    S364_M_FRT_PNL_제품감지_유 AT %MW2002.12 : BOOL;
    S364_M_FRT_PNL_제품감지_이상 AT %MW2014.3 : BOOL;
    S364_M_FRT_RACK_제품감지_무 AT %MW2002.7 : BOOL;
    S364_M_FRT_RACK_제품감지_유 AT %MW2002.6 : BOOL;
    S364_M_FRT_RACK_제품감지_이상 AT %MW2014.0 : BOOL;
    S364_M_LC_정상 AT %MW2007.5 : BOOL; (* S364_M_LC_정상 *)
    S364_M_LH_CB_OFF AT %MW2021.1 : BOOL; (* S364_M_LH_CB_OFF *)
    S364_M_LH_CP_OFF AT %MW2017.0 : BOOL; (* S364_M_LH_CP_OFF *)
    S364_M_LH_INV_이상 AT %MW2019.0 : BOOL; (* S364_M_LH_INV_이상 *)
    S364_M_LH_MC_이상 AT %MW2023.0 : BOOL; (* S364_M_LH_MC_이상 *)
    S364_M_LH_NFB_OFF AT %MW2021.0 : BOOL; (* S364_M_LH_NFB_OFF *)
    S364_M_LH_공기압_이상 AT %MW2013.0 : BOOL; (* S364_M_LH_공기압_이상 *)
    S364_M_MAT_정상 AT %MW2007.6 : BOOL; (* S364_M_MAT_정상 *)
    S364_M_OP_ESTOP_NORMAL AT %MW2007.1 : BOOL; (* S364_M_OP_ESTOP_NORMAL *)
    S364_M_OP_LC_이상 AT %MW2012.0 : BOOL; (* S364_M_OP_LC_이상 *)
    S364_M_OP_MAT_이상 AT %MW2012.1 : BOOL; (* S364_M_OP_MAT_이상 *)
    S364_M_R361_1_DATA_전송_MEMO AT %MW9012.8 : BOOL; (* S364 M R361 1 DATA 전송 MEMO *)
    S364_M_R361_1_DATA_전송_PLS AT %MW9012.9 : BOOL; (* S364 M R361 1 DATA 전송 PLS *)
    S364_M_R361_1_DATA_전송_SIGN AT %MW9012.10 : BOOL; (* S364 M R361 1 DATA 전송 SIGN *)
    S364_M_R361_1_DATA_전송_완료 AT %MW9012.11 : BOOL; (* S364 M R361 1 DATA 전송 완료 *)
    S364_M_R361_1_언로딩완료 AT %MW2001.4 : BOOL;
    S364_M_R361_2_로딩가능 AT %MW2004.9 : BOOL;
    S364_M_R361_2_로딩완료 AT %MW2001.2 : BOOL;
    S364_M_R364_1_용접가능 AT %MW2004.10 : BOOL;
    S364_M_R364_1_용접완료 AT %MW2001.3 : BOOL;
    S364_M_RH_CB_OFF AT %MW2021.4 : BOOL; (* S364_M_RH_CB_OFF *)
    S364_M_RH_CP_OFF AT %MW2017.1 : BOOL; (* S364_M_RH_CP_OFF *)
    S364_M_RH_INV_이상 AT %MW2019.1 : BOOL; (* S364_M_RH_INV_이상 *)
    S364_M_RH_MC_이상 AT %MW2023.1 : BOOL; (* S364_M_RH_MC_이상 *)
    S364_M_RH_NFB_OFF AT %MW2021.3 : BOOL; (* S364_M_RH_NFB_OFF *)
    S364_M_RH_공기압_이상 AT %MW2013.1 : BOOL; (* S364_M_RH_공기압_이상 *)
    S364_M_RR_PNL_제품감지_무 AT %MW2002.15 : BOOL;
    S364_M_RR_PNL_제품감지_유 AT %MW2002.14 : BOOL;
    S364_M_RR_PNL_제품감지_이상 AT %MW2014.4 : BOOL;
    S364_M_RR_RACK_제품감지_무 AT %MW2002.11 : BOOL;
    S364_M_RR_RACK_제품감지_유 AT %MW2002.10 : BOOL;
    S364_M_RR_RACK_제품감지_이상 AT %MW2014.2 : BOOL;
    S364_M_S102_간섭무 AT %MW2004.2 : BOOL; (* S364_M_S102_간섭무 *)
    S364_M_SAFETY_불간섭 AT %MW2004.4 : BOOL; (* S364_M_SAFETY_불간섭 *)
    S364_M_SEMI_자동모드 AT %MW2000.2 : BOOL; (* S364_M_SEMI_자동모드 *)
    S364_M_SEQ AT %MW10120 : WORD; (* S364 M SEQ *)
    S364_M_VIN_NO_1_2 AT %MW10131 : WORD; (* S364 M VIN NO 1 2 *)
    S364_M_VIN_NO_3_4 AT %MW10132 : WORD; (* S364 M VIN NO 3 4 *)
    S364_M_VIN_NO_5_6 AT %MW10133 : WORD; (* S364 M VIN NO 5 6 *)
    S364_M_VIN_NO_7_8 AT %MW10134 : WORD; (* S364 M VIN NO 7 8 *)
    S364_M_VIN_NO_9_10 AT %MW10135 : WORD; (* S364 M VIN NO 9 10 *)
    S364_M_공정_SAFETY_NORMAL AT %MW2007.7 : BOOL; (* S364_M_공정_SAFETY_NORMAL *)
    S364_M_공정_불간섭 AT %MW2004.1 : BOOL; (* S364_M_공정_불간섭 *)
    S364_M_공정_원위치 AT %MW2004.0 : BOOL; (* S364_M_공정_원위치 *)
    S364_M_공정_제품감지_무 AT %MW2002.5 : BOOL; (* S364_M_공정_제품감지_무 *)
    S364_M_공정_제품감지_유 AT %MW2002.4 : BOOL; (* S364_M_공정_제품감지_유 *)
    S364_M_공정_차종_AX AT %MW2002.3 : BOOL; (* S364_M_공정_차종_AX *)
    S364_M_공정_차종_무 AT %MW2002.1 : BOOL; (* S364_M_공정_차종_무 *)
    S364_M_공정_차종_보조 AT %MW2002.2 : BOOL; (* S364_M_공정_차종_보조 *)
    S364_M_공정_차종_유 AT %MW2002.0 : BOOL; (* S364_M_공정_차종_유 *)
    S364_M_동작_선택_1 AT %MW2040.0 : BOOL; (* S364_M_동작_선택_1 *)
    S364_M_동작_선택_10 AT %MW2040.9 : BOOL; (* S364_M_동작_선택_10 *)
    S364_M_동작_선택_11 AT %MW2040.10 : BOOL; (* S364_M_동작_선택_11 *)
    S364_M_동작_선택_12 AT %MW2040.11 : BOOL; (* S364_M_동작_선택_12 *)
    S364_M_동작_선택_13 AT %MW2040.12 : BOOL; (* S364_M_동작_선택_13 *)
    S364_M_동작_선택_14 AT %MW2040.13 : BOOL; (* S364_M_동작_선택_14 *)
    S364_M_동작_선택_15 AT %MW2040.14 : BOOL; (* S364_M_동작_선택_15 *)
    S364_M_동작_선택_16 AT %MW2040.15 : BOOL; (* S364_M_동작_선택_16 *)
    S364_M_동작_선택_17 AT %MW2041.0 : BOOL; (* S364_M_동작_선택_17 *)
    S364_M_동작_선택_18 AT %MW2041.1 : BOOL; (* S364_M_동작_선택_18 *)
    S364_M_동작_선택_19 AT %MW2041.2 : BOOL; (* S364_M_동작_선택_19 *)
    S364_M_동작_선택_2 AT %MW2040.1 : BOOL; (* S364_M_동작_선택_2 *)
    S364_M_동작_선택_20 AT %MW2041.3 : BOOL; (* S364_M_동작_선택_20 *)
    S364_M_동작_선택_21 AT %MW2041.4 : BOOL; (* S364_M_동작_선택_21 *)
    S364_M_동작_선택_22 AT %MW2041.5 : BOOL; (* S364_M_동작_선택_22 *)
    S364_M_동작_선택_23 AT %MW2041.6 : BOOL; (* S364_M_동작_선택_23 *)
    S364_M_동작_선택_24 AT %MW2041.7 : BOOL; (* S364_M_동작_선택_24 *)
    S364_M_동작_선택_25 AT %MW2041.8 : BOOL; (* S364_M_동작_선택_25 *)
    S364_M_동작_선택_26 AT %MW2041.9 : BOOL; (* S364_M_동작_선택_26 *)
    S364_M_동작_선택_27 AT %MW2041.10 : BOOL; (* S364_M_동작_선택_27 *)
    S364_M_동작_선택_28 AT %MW2041.11 : BOOL; (* S364_M_동작_선택_28 *)
    S364_M_동작_선택_29 AT %MW2041.12 : BOOL; (* S364_M_동작_선택_29 *)
    S364_M_동작_선택_3 AT %MW2040.2 : BOOL; (* S364_M_동작_선택_3 *)
    S364_M_동작_선택_30 AT %MW2041.13 : BOOL; (* S364_M_동작_선택_30 *)
    S364_M_동작_선택_31 AT %MW2041.14 : BOOL; (* S364_M_동작_선택_31 *)
    S364_M_동작_선택_32 AT %MW2041.15 : BOOL; (* S364_M_동작_선택_32 *)
    S364_M_동작_선택_4 AT %MW2040.3 : BOOL; (* S364_M_동작_선택_4 *)
    S364_M_동작_선택_5 AT %MW2040.4 : BOOL; (* S364_M_동작_선택_5 *)
    S364_M_동작_선택_6 AT %MW2040.5 : BOOL; (* S364_M_동작_선택_6 *)
    S364_M_동작_선택_7 AT %MW2040.6 : BOOL; (* S364_M_동작_선택_7 *)
    S364_M_동작_선택_8 AT %MW2040.7 : BOOL; (* S364_M_동작_선택_8 *)
    S364_M_동작_선택_9 AT %MW2040.8 : BOOL; (* S364_M_동작_선택_9 *)
    S364_M_부저_정지_보조 AT %MW2000.11 : BOOL; (* S364_M_부저_정지_보조 *)
    S364_M_수동모드 AT %MW2000.3 : BOOL; (* S364 선택 수동모드 *)
    S364_M_운전준비_ON AT %MW2000.0 : BOOL; (* S364 운전준비 ON *)
    S364_M_이상_리셋_보조 AT %MW2000.10 : BOOL; (* S364_M_이상_리셋_보조 *)
    S364_M_자동_START AT %MW2000.5 : BOOL; (* S364 자동운전중 *)
    S364_M_자동_운전중 AT %MW2000.4 : BOOL; (* S364 자동운전중 *)
    S364_M_자동모드 AT %MW2000.1 : BOOL; (* S364 선택 자동모드 *)
    S364_M_작업_완료 AT %MW2001.0 : BOOL; (* S364_M_작업_완료 *)
    S364_M_작업완료_SET_PLS AT %MW2000.8 : BOOL; (* S364 M 작업완료 SET PLS *)
    S364_M_작업완료_리셋_PLS AT %MW2000.9 : BOOL; (* S364 M 작업완료 리셋 PLS *)
    S364_M_작업자_작업가능 AT %MW2004.8 : BOOL;
    S364_M_작업자_작업완료 AT %MW2001.1 : BOOL;
    S364_M_전체_용접완료 AT %MW2006.0 : BOOL;
    S364_M_차종1_AX AT %MW10121.0 : BOOL; (* S364 M 차종1 AX *)
    S364_M_차종1_B AT %MW10121.1 : BOOL; (* S364 M 차종1 B *)
    S364_M_차종1_C AT %MW10121.2 : BOOL; (* S364 M 차종1 C *)
    S364_M_차종1_D AT %MW10121.3 : BOOL; (* S364 M 차종1 D *)
    S364_M_차종1_E AT %MW10121.4 : BOOL; (* S364 M 차종1 E *)
    S364_M_차종1_F AT %MW10121.5 : BOOL; (* S364 M 차종1 F *)
    S364_M_차종1_G AT %MW10121.6 : BOOL; (* S364 M 차종1 G *)
    S364_M_차종1_H AT %MW10121.7 : BOOL; (* S364 M 차종1 H *)
    S364_M_차종2_3DR AT %MW10121.8 : BOOL; (* S364 M 차종2 3DR *)
    S364_M_차종2_4DR AT %MW10121.9 : BOOL; (* S364 M 차종2 4DR *)
    S364_M_차종2_5DR AT %MW10121.10 : BOOL; (* S364 M 차종2 5DR *)
    S364_M_차종2_SP1 AT %MW10121.12 : BOOL; (* S364 M 차종2 SP1 *)
    S364_M_차종2_SP2 AT %MW10121.13 : BOOL; (* S364 M 차종2 SP2 *)
    S364_M_차종2_WGN AT %MW10121.11 : BOOL; (* S364 M 차종2 WGN *)
    S364_M_차종3_LHD AT %MW10121.14 : BOOL; (* S364 M 차종3 LHD *)
    S364_M_차종3_RHD AT %MW10121.15 : BOOL; (* S364 M 차종3 RHD *)
    S364_M_차종4_EEC AT %MW10122.3 : BOOL; (* S364 M 차종4 EEC *)
    S364_M_차종4_SP1 AT %MW10122.8 : BOOL; (* S364 M 차종4 SP1 *)
    S364_M_차종4_SP2 AT %MW10122.9 : BOOL; (* S364 M 차종4 SP2 *)
    S364_M_차종4_SP3 AT %MW10122.11 : BOOL; (* S364 M 차종4 SP3 *)
    S364_M_차종4_SP4 AT %MW10122.12 : BOOL; (* S364 M 차종4 SP4 *)
    S364_M_차종4_SP5 AT %MW10122.13 : BOOL; (* S364 M 차종4 SP5 *)
    S364_M_차종4_SP6 AT %MW10122.14 : BOOL; (* S364 M 차종4 SP6 *)
    S364_M_차종4_SP7 AT %MW10122.15 : BOOL; (* S364 M 차종4 SP7 *)
    S364_M_차종4_내수 AT %MW10122.0 : BOOL; (* S364 M 차종4 내수 *)
    S364_M_차종4_러시아 AT %MW10122.10 : BOOL; (* S364 M 차종4 러시아 *)
    S364_M_차종4_북미 AT %MW10122.2 : BOOL; (* S364 M 차종4 북미 *)
    S364_M_차종4_브라질 AT %MW10122.7 : BOOL; (* S364 M 차종4 브라질 *)
    S364_M_차종4_수출 AT %MW10122.1 : BOOL; (* S364 M 차종4 수출 *)
    S364_M_차종4_중국 AT %MW10122.6 : BOOL; (* S364 M 차종4 중국 *)
    S364_M_차종4_중동 AT %MW10122.5 : BOOL; (* S364 M 차종4 중동 *)
    S364_M_차종4_호주 AT %MW10122.4 : BOOL; (* S364 M 차종4 호주 *)
    S364_M_차종5_AT AT %MW10123.1 : BOOL; (* S364 M 차종5 AT *)
    S364_M_차종5_MT AT %MW10123.0 : BOOL; (* S364 M 차종5 MT *)
    S364_M_차종5_SP1 AT %MW10123.2 : BOOL; (* S364 M 차종5 SP1 *)
    S364_M_차종6_DSROOF AT %MW10123.6 : BOOL; (* S364 M 차종6 DSROOF *)
    S364_M_차종6_SP1 AT %MW10123.7 : BOOL; (* S364 M 차종6 SP1 *)
    S364_M_차종6_썬루프 AT %MW10123.4 : BOOL; (* S364 M 차종6 썬루프 *)
    S364_M_차종6_일반루프 AT %MW10123.3 : BOOL; (* S364 M 차종6 일반루프 *)
    S364_M_차종6_파노라마루프 AT %MW10123.5 : BOOL; (* S364 M 차종6 파노라마루프 *)
    S364_M_차종7_DSL AT %MW10123.9 : BOOL; (* S364 M 차종7 DSL *)
    S364_M_차종7_GSL AT %MW10123.8 : BOOL; (* S364 M 차종7 GSL *)
    S364_M_차종7_SP1 AT %MW10123.10 : BOOL; (* S364 M 차종7 SP1 *)
    S364_M_차종7_SP2 AT %MW10123.11 : BOOL; (* S364 M 차종7 SP2 *)
    S364_M_차종7_SP3 AT %MW10123.12 : BOOL; (* S364 M 차종7 SP3 *)
    S364_M_차종7_SP4 AT %MW10123.13 : BOOL; (* S364 M 차종7 SP4 *)
    S364_M_차종7_SP5 AT %MW10123.14 : BOOL; (* S364 M 차종7 SP5 *)
    S364_M_차종7_SP6 AT %MW10123.15 : BOOL; (* S364 M 차종7 SP6 *)
    S364_M_차종8_2WD AT %MW10124.0 : BOOL; (* S364 M 차종8 2WD *)
    S364_M_차종8_4WD AT %MW10124.1 : BOOL; (* S364 M 차종8 4WD *)
    S364_M_차종8_SP1 AT %MW10124.2 : BOOL; (* S364 M 차종8 SP1 *)
    S364_M_차종9_MPI AT %MW10124.3 : BOOL; (* S364 M 차종9 MPI *)
    S364_M_차종9_SP1 AT %MW10124.5 : BOOL; (* S364 M 차종9 SP1 *)
    S364_M_차종9_SP10 AT %MW10124.14 : BOOL; (* S364 M 차종9 SP10 *)
    S364_M_차종9_SP11 AT %MW10124.15 : BOOL; (* S364 M 차종9 SP11 *)
    S364_M_차종9_SP2 AT %MW10124.6 : BOOL; (* S364 M 차종9 SP2 *)
    S364_M_차종9_SP3 AT %MW10124.7 : BOOL; (* S364 M 차종9 SP3 *)
    S364_M_차종9_SP4 AT %MW10124.8 : BOOL; (* S364 M 차종9 SP4 *)
    S364_M_차종9_SP5 AT %MW10124.9 : BOOL; (* S364 M 차종9 SP5 *)
    S364_M_차종9_SP6 AT %MW10124.10 : BOOL; (* S364 M 차종9 SP6 *)
    S364_M_차종9_SP7 AT %MW10124.11 : BOOL; (* S364 M 차종9 SP7 *)
    S364_M_차종9_SP8 AT %MW10124.12 : BOOL; (* S364 M 차종9 SP8 *)
    S364_M_차종9_SP9 AT %MW10124.13 : BOOL; (* S364 M 차종9 SP9 *)
    S364_M_차종9_T_GDI AT %MW10124.4 : BOOL; (* S364 M 차종9 T GDI *)
    S364_M_차종_AS AT %MW10130.9 : BOOL; (* S364 M 차종 AS *)
    S364_M_차종_OPT1_R_RACK_무 AT %MW10125.3 : BOOL; (* S364 M 차종 OPT1 R RACK 무 *)
    S364_M_차종_OPT1_R_RACK_유 AT %MW10125.2 : BOOL; (* S364 M 차종 OPT1 R RACK 유 *)
    S364_M_차종_OPT1_SP1 AT %MW10125.10 : BOOL; (* S364 M 차종 OPT1 SP1 *)
    S364_M_차종_OPT1_SP2 AT %MW10125.11 : BOOL; (* S364 M 차종 OPT1 SP2 *)
    S364_M_차종_OPT1_SP3 AT %MW10125.12 : BOOL; (* S364 M 차종 OPT1 SP3 *)
    S364_M_차종_OPT1_SP4 AT %MW10125.13 : BOOL; (* S364 M 차종 OPT1 SP4 *)
    S364_M_차종_OPT1_SP5 AT %MW10125.14 : BOOL; (* S364 M 차종 OPT1 SP5 *)
    S364_M_차종_OPT1_SP6 AT %MW10125.15 : BOOL; (* S364 M 차종 OPT1 SP6 *)
    S364_M_차종_OPT1_S_REP_EATER_무 AT %MW10125.7 : BOOL; (* S364 M 차종 OPT1 S REP EATER 무 *)
    S364_M_차종_OPT1_S_REP_EATER_유 AT %MW10125.6 : BOOL; (* S364 M 차종 OPT1 S REP EATER 유 *)
    S364_M_차종_OPT1_VAN_무 AT %MW10125.9 : BOOL; (* S364 M 차종 OPT1 VAN 무 *)
    S364_M_차종_OPT1_VAN_유 AT %MW10125.8 : BOOL; (* S364 M 차종 OPT1 VAN 유 *)
    S364_M_차종_OPT1_슬라이딩_무 AT %MW10125.1 : BOOL; (* S364 M 차종 OPT1 슬라이딩 무 *)
    S364_M_차종_OPT1_슬라이딩_유 AT %MW10125.0 : BOOL; (* S364 M 차종 OPT1 슬라이딩 유 *)
    S364_M_차종_OPT1_폴딩_무 AT %MW10125.5 : BOOL; (* S364 M 차종 OPT1 폴딩 무 *)
    S364_M_차종_OPT1_폴딩_유 AT %MW10125.4 : BOOL; (* S364 M 차종 OPT1 폴딩 유 *)
    S364_M_차종_OPT2_SP_WORD1 AT %MW10126 : WORD; (* S364 M 차종 OPT2 SP WORD1 *)
    S364_M_차종_OPT3_SP_WORD2 AT %MW10127 : WORD; (* S364 M 차종 OPT3 SP WORD2 *)
    S364_M_차종_OPT4_SP_WORD3 AT %MW10128 : WORD; (* S364 M 차종 OPT4 SP WORD3 *)
    S364_M_차종_OPT5_SP_WORD4 AT %MW10129 : WORD; (* S364 M 차종 OPT5 SP WORD4 *)
    S364_M_차종_SP1 AT %MW10130.0 : BOOL; (* S364 M 차종 SP1 *)
    S364_M_차종_SP2 AT %MW10130.1 : BOOL; (* S364 M 차종 SP2 *)
    S364_M_차종_SP3 AT %MW10130.2 : BOOL; (* S364 M 차종 SP3 *)
    S364_M_차종_SP4 AT %MW10130.3 : BOOL; (* S364 M 차종 SP4 *)
    S364_M_차종_SP5 AT %MW10130.4 : BOOL; (* S364 M 차종 SP5 *)
    S364_M_차종_SP6 AT %MW10130.5 : BOOL; (* S364 M 차종 SP6 *)
    S364_M_차종_SP7 AT %MW10130.6 : BOOL; (* S364 M 차종 SP7 *)
    S364_M_차종_SP8 AT %MW10130.7 : BOOL; (* S364 M 차종 SP8 *)
    S364_M_차종_SP9 AT %MW10130.15 : BOOL; (* S364 M 차종 SP9 *)
    S364_M_차종_공대차 AT %MW10130.12 : BOOL; (* S364 M 차종 공대차 *)
    S364_M_차종_공차 AT %MW10130.10 : BOOL; (* S364 M 차종 공차 *)
    S364_M_차종_불량대차 AT %MW10130.13 : BOOL; (* S364 M 차종 불량대차 *)
    S364_M_차종_불량차 AT %MW10130.11 : BOOL; (* S364 M 차종 불량차 *)
    S364_M_차종_비축 AT %MW10130.8 : BOOL; (* S364 M 차종 비축 *)
    S364_M_차종_취출대차 AT %MW10130.14 : BOOL; (* S364 M 차종 취출대차 *)
    S364_M_총괄_CP_이상 AT %MW2009.7 : BOOL; (* S364 CP OFF 이상 *)
    S364_M_총괄_CT_이상 AT %MW2010.4 : BOOL; (* S364   TACK TIME 이상 *)
    S364_M_총괄_EOCR_이상 AT %MW2009.8 : BOOL; (* S364_M_총괄_EOCR_이상 *)
    S364_M_총괄_INV_이상 AT %MW2009.9 : BOOL; (* S364_M_총괄_INV_이상 *)
    S364_M_총괄_LS_이상 AT %MW2009.15 : BOOL; (* S364 LS 이상 *)
    S364_M_총괄_MATCH_이상 AT %MW2010.0 : BOOL; (* S364 매트SW 이상 *)
    S364_M_총괄_MC_이상 AT %MW2009.13 : BOOL; (* S364_M_총괄_MC_이상 *)
    S364_M_총괄_MOTOR_이상 AT %MW2010.3 : BOOL; (* S364_M_총괄_MOTOR_이상 *)
    S364_M_총괄_NFB_이상 AT %MW2009.11 : BOOL; (* S364_M_총괄_NFB_이상 *)
    S364_M_총괄_ROBOT_이상 AT %MW2010.1 : BOOL; (* S364 ROBOT 이상 *)
    S364_M_총괄_SAFETY_이상 AT %MW2009.2 : BOOL; (* S364 SAFETY 이상 *)
    S364_M_총괄_SRV_이상 AT %MW2009.10 : BOOL; (* S364_M_총괄_SRV_이상 *)
    S364_M_총괄_공기압_이상 AT %MW2009.3 : BOOL; (* S364 공기압 이상 *)
    S364_M_총괄_비상정지_이상 AT %MW2009.1 : BOOL; (* S364_M_총괄_비상정지_이상 *)
    S364_M_총괄_사양_이상 AT %MW2009.6 : BOOL; (* S364 사양 이상 *)
    S364_M_총괄_오버런_이상 AT %MW2009.12 : BOOL; (* S364_M_총괄_오버런_이상 *)
    S364_M_총괄_용접타점수_이상 AT %MW2010.2 : BOOL; (* S364 용접타점수 이상 *)
    S364_M_총괄_이상 AT %MW2009.0 : BOOL; (* S364_M_총괄_이상 *)
    S364_M_총괄_제품감지_이상 AT %MW2009.4 : BOOL; (* S364 제품감지 이상 *)
    S364_M_총괄_차종_이상 AT %MW2009.5 : BOOL; (* S364 차종 이상 *)
    S364_M_총괄_통신_이상 AT %MW2009.14 : BOOL; (* S364 통신이상 *)
    S364_RH_M_NODE_7_15_통신_이상 AT %MW2024.1 : BOOL;
    S364_전진_ON AT %MW2048.1 : BOOL; (* S364_전진_ON *)
    S364_후진_ON AT %MW2048.2 : BOOL; (* S364_후진_ON *)
    S365_HOME AT %MW2548.0 : BOOL; (* S365_HOME *)
    S365_M_BYPASS_보조 AT %MW2503.15 : BOOL; (* S365 M BYPASS 보조 *)
    S365_M_CTIME_OVER_ALRAM AT %MW2507.14 : BOOL; (* S365_M_CTIME_OVER_ALRAM *)
    S365_M_CTIME_OVER_MUTE AT %MW2507.13 : BOOL; (* S365_M_CTIME_OVER_MUTE *)
    S365_M_DATA_삭제_PLS AT %MW9013.0 : BOOL; (* S365 M DATA 삭제 PLS *)
    S365_M_DATA_삭제_SIGN AT %MW9013.1 : BOOL; (* S365 M DATA 삭제 SIGN *)
    S365_M_DATA_삭제_완료 AT %MW9013.2 : BOOL; (* S365 M DATA 삭제 완료 *)
    S365_M_LC_정상 AT %MW2507.5 : BOOL; (* S365_M_LC_정상 *)
    S365_M_MAT_정상 AT %MW2507.6 : BOOL; (* S365_M_MAT_정상 *)
    S365_M_NODE_6_01_통신_이상 AT %MW2524.0 : BOOL;
    S365_M_OP_ESTOP_NORMAL AT %MW2507.1 : BOOL; (* S365_M_OP_ESTOP_NORMAL *)
    S365_M_R361_1_안착완료 AT %MW2501.1 : BOOL;
    S365_M_R361_1_언로딩완료 AT %MW2501.2 : BOOL;
    S365_M_S102_간섭무 AT %MW2504.2 : BOOL; (* S365_M_S102_간섭무 *)
    S365_M_S361_1_DATA_전송_MEMO AT %MW9013.8 : BOOL; (* S365 M S361 1 DATA 전송 MEMO *)
    S365_M_S361_1_DATA_전송_PLS AT %MW9013.9 : BOOL; (* S365 M S361 1 DATA 전송 PLS *)
    S365_M_S361_1_DATA_전송_SIGN AT %MW9013.10 : BOOL; (* S365 M S361 1 DATA 전송 SIGN *)
    S365_M_S361_1_DATA_전송_완료 AT %MW9013.11 : BOOL; (* S365 M S361 1 DATA 전송 완료 *)
    S365_M_SAFETY_불간섭 AT %MW2504.4 : BOOL; (* S365_M_SAFETY_불간섭 *)
    S365_M_SEMI_자동모드 AT %MW2500.2 : BOOL; (* S365_M_SEMI_자동모드 *)
    S365_M_SEQ AT %MW10140 : WORD; (* S365 M SEQ *)
    S365_M_VIN_NO_1_2 AT %MW10151 : WORD; (* S365 M VIN NO 1 2 *)
    S365_M_VIN_NO_3_4 AT %MW10152 : WORD; (* S365 M VIN NO 3 4 *)
    S365_M_VIN_NO_5_6 AT %MW10153 : WORD; (* S365 M VIN NO 5 6 *)
    S365_M_VIN_NO_7_8 AT %MW10154 : WORD; (* S365 M VIN NO 7 8 *)
    S365_M_VIN_NO_9_10 AT %MW10155 : WORD; (* S365 M VIN NO 9 10 *)
    S365_M_공정_SAFETY_NORMAL AT %MW2507.7 : BOOL; (* S365_M_공정_SAFETY_NORMAL *)
    S365_M_공정_불간섭 AT %MW2504.1 : BOOL; (* S365_M_공정_불간섭 *)
    S365_M_공정_원위치 AT %MW2504.0 : BOOL; (* S365_M_공정_원위치 *)
    S365_M_공정_제품감지_무 AT %MW2501.4 : BOOL; (* S365_M_공정_제품감지_무 *)
    S365_M_공정_제품감지_유 AT %MW2501.3 : BOOL; (* S365_M_공정_제품감지_유 *)
    S365_M_공정_차종_무 AT %MW2502.1 : BOOL; (* S365_M_공정_차종_무 *)
    S365_M_공정_차종_보조 AT %MW2502.2 : BOOL; (* S365_M_공정_차종_보조 *)
    S365_M_공정_차종_유 AT %MW2502.0 : BOOL; (* S365_M_공정_차종_유 *)
    S365_M_동작_선택_1 AT %MW2540.0 : BOOL; (* S365_M_동작_선택_1 *)
    S365_M_동작_선택_10 AT %MW2540.9 : BOOL; (* S365_M_동작_선택_10 *)
    S365_M_동작_선택_11 AT %MW2540.10 : BOOL; (* S365_M_동작_선택_11 *)
    S365_M_동작_선택_12 AT %MW2540.11 : BOOL; (* S365_M_동작_선택_12 *)
    S365_M_동작_선택_13 AT %MW2540.12 : BOOL; (* S365_M_동작_선택_13 *)
    S365_M_동작_선택_14 AT %MW2540.13 : BOOL; (* S365_M_동작_선택_14 *)
    S365_M_동작_선택_15 AT %MW2540.14 : BOOL; (* S365_M_동작_선택_15 *)
    S365_M_동작_선택_16 AT %MW2540.15 : BOOL; (* S365_M_동작_선택_16 *)
    S365_M_동작_선택_17 AT %MW2541.0 : BOOL; (* S365_M_동작_선택_17 *)
    S365_M_동작_선택_18 AT %MW2541.1 : BOOL; (* S365_M_동작_선택_18 *)
    S365_M_동작_선택_19 AT %MW2541.2 : BOOL; (* S365_M_동작_선택_19 *)
    S365_M_동작_선택_2 AT %MW2540.1 : BOOL; (* S365_M_동작_선택_2 *)
    S365_M_동작_선택_20 AT %MW2541.3 : BOOL; (* S365_M_동작_선택_20 *)
    S365_M_동작_선택_21 AT %MW2541.4 : BOOL; (* S365_M_동작_선택_21 *)
    S365_M_동작_선택_22 AT %MW2541.5 : BOOL; (* S365_M_동작_선택_22 *)
    S365_M_동작_선택_23 AT %MW2541.6 : BOOL; (* S365_M_동작_선택_23 *)
    S365_M_동작_선택_24 AT %MW2541.7 : BOOL; (* S365_M_동작_선택_24 *)
    S365_M_동작_선택_25 AT %MW2541.8 : BOOL; (* S365_M_동작_선택_25 *)
    S365_M_동작_선택_26 AT %MW2541.9 : BOOL; (* S365_M_동작_선택_26 *)
    S365_M_동작_선택_27 AT %MW2541.10 : BOOL; (* S365_M_동작_선택_27 *)
    S365_M_동작_선택_28 AT %MW2541.11 : BOOL; (* S365_M_동작_선택_28 *)
    S365_M_동작_선택_29 AT %MW2541.12 : BOOL; (* S365_M_동작_선택_29 *)
    S365_M_동작_선택_3 AT %MW2540.2 : BOOL; (* S365_M_동작_선택_3 *)
    S365_M_동작_선택_30 AT %MW2541.13 : BOOL; (* S365_M_동작_선택_30 *)
    S365_M_동작_선택_31 AT %MW2541.14 : BOOL; (* S365_M_동작_선택_31 *)
    S365_M_동작_선택_32 AT %MW2541.15 : BOOL; (* S365_M_동작_선택_32 *)
    S365_M_동작_선택_4 AT %MW2540.3 : BOOL; (* S365_M_동작_선택_4 *)
    S365_M_동작_선택_5 AT %MW2540.4 : BOOL; (* S365_M_동작_선택_5 *)
    S365_M_동작_선택_6 AT %MW2540.5 : BOOL; (* S365_M_동작_선택_6 *)
    S365_M_동작_선택_7 AT %MW2540.6 : BOOL; (* S365_M_동작_선택_7 *)
    S365_M_동작_선택_8 AT %MW2540.7 : BOOL; (* S365_M_동작_선택_8 *)
    S365_M_동작_선택_9 AT %MW2540.8 : BOOL; (* S365_M_동작_선택_9 *)
    S365_M_부저_정지_보조 AT %MW2500.11 : BOOL; (* S365_M_부저_정지_보조 *)
    S365_M_수동모드 AT %MW2500.3 : BOOL; (* S365 선택 수동모드 *)
    S365_M_운전준비_ON AT %MW2500.0 : BOOL; (* S365 운전준비 ON *)
    S365_M_이상_리셋_보조 AT %MW2500.10 : BOOL; (* S365_M_이상_리셋_보조 *)
    S365_M_자동_START AT %MW2500.5 : BOOL; (* S365 자동운전중 *)
    S365_M_자동_운전중 AT %MW2500.4 : BOOL; (* S365 자동운전중 *)
    S365_M_자동모드 AT %MW2500.1 : BOOL; (* S365 선택 자동모드 *)
    S365_M_작업_완료 AT %MW2501.0 : BOOL; (* S365_M_작업_완료 *)
    S365_M_작업완료_SET_PLS AT %MW2500.8 : BOOL; (* S365 M 작업완료 SET PLS *)
    S365_M_작업완료_리셋_PLS AT %MW2500.9 : BOOL; (* S365 M 작업완료 리셋 PLS *)
    S365_M_차종1_AX AT %MW10141.0 : BOOL; (* S365 M 차종1 AX *)
    S365_M_차종1_B AT %MW10141.1 : BOOL; (* S365 M 차종1 B *)
    S365_M_차종1_C AT %MW10141.2 : BOOL; (* S365 M 차종1 C *)
    S365_M_차종1_D AT %MW10141.3 : BOOL; (* S365 M 차종1 D *)
    S365_M_차종1_E AT %MW10141.4 : BOOL; (* S365 M 차종1 E *)
    S365_M_차종1_F AT %MW10141.5 : BOOL; (* S365 M 차종1 F *)
    S365_M_차종1_G AT %MW10141.6 : BOOL; (* S365 M 차종1 G *)
    S365_M_차종1_H AT %MW10141.7 : BOOL; (* S365 M 차종1 H *)
    S365_M_차종2_3DR AT %MW10141.8 : BOOL; (* S365 M 차종2 3DR *)
    S365_M_차종2_4DR AT %MW10141.9 : BOOL; (* S365 M 차종2 4DR *)
    S365_M_차종2_5DR AT %MW10141.10 : BOOL; (* S365 M 차종2 5DR *)
    S365_M_차종2_SP1 AT %MW10141.12 : BOOL; (* S365 M 차종2 SP1 *)
    S365_M_차종2_SP2 AT %MW10141.13 : BOOL; (* S365 M 차종2 SP2 *)
    S365_M_차종2_WGN AT %MW10141.11 : BOOL; (* S365 M 차종2 WGN *)
    S365_M_차종3_LHD AT %MW10141.14 : BOOL; (* S365 M 차종3 LHD *)
    S365_M_차종3_RHD AT %MW10141.15 : BOOL; (* S365 M 차종3 RHD *)
    S365_M_차종4_EEC AT %MW10142.3 : BOOL; (* S365 M 차종4 EEC *)
    S365_M_차종4_SP1 AT %MW10142.8 : BOOL; (* S365 M 차종4 SP1 *)
    S365_M_차종4_SP2 AT %MW10142.9 : BOOL; (* S365 M 차종4 SP2 *)
    S365_M_차종4_SP3 AT %MW10142.11 : BOOL; (* S365 M 차종4 SP3 *)
    S365_M_차종4_SP4 AT %MW10142.12 : BOOL; (* S365 M 차종4 SP4 *)
    S365_M_차종4_SP5 AT %MW10142.13 : BOOL; (* S365 M 차종4 SP5 *)
    S365_M_차종4_SP6 AT %MW10142.14 : BOOL; (* S365 M 차종4 SP6 *)
    S365_M_차종4_SP7 AT %MW10142.15 : BOOL; (* S365 M 차종4 SP7 *)
    S365_M_차종4_내수 AT %MW10142.0 : BOOL; (* S365 M 차종4 내수 *)
    S365_M_차종4_러시아 AT %MW10142.10 : BOOL; (* S365 M 차종4 러시아 *)
    S365_M_차종4_북미 AT %MW10142.2 : BOOL; (* S365 M 차종4 북미 *)
    S365_M_차종4_브라질 AT %MW10142.7 : BOOL; (* S365 M 차종4 브라질 *)
    S365_M_차종4_수출 AT %MW10142.1 : BOOL; (* S365 M 차종4 수출 *)
    S365_M_차종4_중국 AT %MW10142.6 : BOOL; (* S365 M 차종4 중국 *)
    S365_M_차종4_중동 AT %MW10142.5 : BOOL; (* S365 M 차종4 중동 *)
    S365_M_차종4_호주 AT %MW10142.4 : BOOL; (* S365 M 차종4 호주 *)
    S365_M_차종5_AT AT %MW10143.1 : BOOL; (* S365 M 차종5 AT *)
    S365_M_차종5_MT AT %MW10143.0 : BOOL; (* S365 M 차종5 MT *)
    S365_M_차종5_SP1 AT %MW10143.2 : BOOL; (* S365 M 차종5 SP1 *)
    S365_M_차종6_DSROOF AT %MW10143.6 : BOOL; (* S365 M 차종6 DSROOF *)
    S365_M_차종6_SP1 AT %MW10143.7 : BOOL; (* S365 M 차종6 SP1 *)
    S365_M_차종6_썬루프 AT %MW10143.4 : BOOL; (* S365 M 차종6 썬루프 *)
    S365_M_차종6_일반루프 AT %MW10143.3 : BOOL; (* S365 M 차종6 일반루프 *)
    S365_M_차종6_파노라마루프 AT %MW10143.5 : BOOL; (* S365 M 차종6 파노라마루프 *)
    S365_M_차종7_DSL AT %MW10143.9 : BOOL; (* S365 M 차종7 DSL *)
    S365_M_차종7_GSL AT %MW10143.8 : BOOL; (* S365 M 차종7 GSL *)
    S365_M_차종7_SP1 AT %MW10143.10 : BOOL; (* S365 M 차종7 SP1 *)
    S365_M_차종7_SP2 AT %MW10143.11 : BOOL; (* S365 M 차종7 SP2 *)
    S365_M_차종7_SP3 AT %MW10143.12 : BOOL; (* S365 M 차종7 SP3 *)
    S365_M_차종7_SP4 AT %MW10143.13 : BOOL; (* S365 M 차종7 SP4 *)
    S365_M_차종7_SP5 AT %MW10143.14 : BOOL; (* S365 M 차종7 SP5 *)
    S365_M_차종7_SP6 AT %MW10143.15 : BOOL; (* S365 M 차종7 SP6 *)
    S365_M_차종8_2WD AT %MW10144.0 : BOOL; (* S365 M 차종8 2WD *)
    S365_M_차종8_4WD AT %MW10144.1 : BOOL; (* S365 M 차종8 4WD *)
    S365_M_차종8_SP1 AT %MW10144.2 : BOOL; (* S365 M 차종8 SP1 *)
    S365_M_차종9_MPI AT %MW10144.3 : BOOL; (* S365 M 차종9 MPI *)
    S365_M_차종9_SP1 AT %MW10144.5 : BOOL; (* S365 M 차종9 SP1 *)
    S365_M_차종9_SP10 AT %MW10144.14 : BOOL; (* S365 M 차종9 SP10 *)
    S365_M_차종9_SP11 AT %MW10144.15 : BOOL; (* S365 M 차종9 SP11 *)
    S365_M_차종9_SP2 AT %MW10144.6 : BOOL; (* S365 M 차종9 SP2 *)
    S365_M_차종9_SP3 AT %MW10144.7 : BOOL; (* S365 M 차종9 SP3 *)
    S365_M_차종9_SP4 AT %MW10144.8 : BOOL; (* S365 M 차종9 SP4 *)
    S365_M_차종9_SP5 AT %MW10144.9 : BOOL; (* S365 M 차종9 SP5 *)
    S365_M_차종9_SP6 AT %MW10144.10 : BOOL; (* S365 M 차종9 SP6 *)
    S365_M_차종9_SP7 AT %MW10144.11 : BOOL; (* S365 M 차종9 SP7 *)
    S365_M_차종9_SP8 AT %MW10144.12 : BOOL; (* S365 M 차종9 SP8 *)
    S365_M_차종9_SP9 AT %MW10144.13 : BOOL; (* S365 M 차종9 SP9 *)
    S365_M_차종9_T_GDI AT %MW10144.4 : BOOL; (* S365 M 차종9 T GDI *)
    S365_M_차종_AS AT %MW10150.9 : BOOL; (* S365 M 차종 AS *)
    S365_M_차종_OPT1_R_RACK_무 AT %MW10145.3 : BOOL; (* S365 M 차종 OPT1 R RACK 무 *)
    S365_M_차종_OPT1_R_RACK_유 AT %MW10145.2 : BOOL; (* S365 M 차종 OPT1 R RACK 유 *)
    S365_M_차종_OPT1_SP1 AT %MW10145.10 : BOOL; (* S365 M 차종 OPT1 SP1 *)
    S365_M_차종_OPT1_SP2 AT %MW10145.11 : BOOL; (* S365 M 차종 OPT1 SP2 *)
    S365_M_차종_OPT1_SP3 AT %MW10145.12 : BOOL; (* S365 M 차종 OPT1 SP3 *)
    S365_M_차종_OPT1_SP4 AT %MW10145.13 : BOOL; (* S365 M 차종 OPT1 SP4 *)
    S365_M_차종_OPT1_SP5 AT %MW10145.14 : BOOL; (* S365 M 차종 OPT1 SP5 *)
    S365_M_차종_OPT1_SP6 AT %MW10145.15 : BOOL; (* S365 M 차종 OPT1 SP6 *)
    S365_M_차종_OPT1_S_REP_EATER_무 AT %MW10145.7 : BOOL; (* S365 M 차종 OPT1 S REP EATER 무 *)
    S365_M_차종_OPT1_S_REP_EATER_유 AT %MW10145.6 : BOOL; (* S365 M 차종 OPT1 S REP EATER 유 *)
    S365_M_차종_OPT1_VAN_무 AT %MW10145.9 : BOOL; (* S365 M 차종 OPT1 VAN 무 *)
    S365_M_차종_OPT1_VAN_유 AT %MW10145.8 : BOOL; (* S365 M 차종 OPT1 VAN 유 *)
    S365_M_차종_OPT1_슬라이딩_무 AT %MW10145.1 : BOOL; (* S365 M 차종 OPT1 슬라이딩 무 *)
    S365_M_차종_OPT1_슬라이딩_유 AT %MW10145.0 : BOOL; (* S365 M 차종 OPT1 슬라이딩 유 *)
    S365_M_차종_OPT1_폴딩_무 AT %MW10145.5 : BOOL; (* S365 M 차종 OPT1 폴딩 무 *)
    S365_M_차종_OPT1_폴딩_유 AT %MW10145.4 : BOOL; (* S365 M 차종 OPT1 폴딩 유 *)
    S365_M_차종_OPT2_SP_WORD1 AT %MW10146 : WORD; (* S365 M 차종 OPT2 SP WORD1 *)
    S365_M_차종_OPT3_SP_WORD2 AT %MW10147 : WORD; (* S365 M 차종 OPT3 SP WORD2 *)
    S365_M_차종_OPT4_SP_WORD3 AT %MW10148 : WORD; (* S365 M 차종 OPT4 SP WORD3 *)
    S365_M_차종_OPT5_SP_WORD4 AT %MW10149 : WORD; (* S365 M 차종 OPT5 SP WORD4 *)
    S365_M_차종_SP1 AT %MW10150.0 : BOOL; (* S365 M 차종 SP1 *)
    S365_M_차종_SP2 AT %MW10150.1 : BOOL; (* S365 M 차종 SP2 *)
    S365_M_차종_SP3 AT %MW10150.2 : BOOL; (* S365 M 차종 SP3 *)
    S365_M_차종_SP4 AT %MW10150.3 : BOOL; (* S365 M 차종 SP4 *)
    S365_M_차종_SP5 AT %MW10150.4 : BOOL; (* S365 M 차종 SP5 *)
    S365_M_차종_SP6 AT %MW10150.5 : BOOL; (* S365 M 차종 SP6 *)
    S365_M_차종_SP7 AT %MW10150.6 : BOOL; (* S365 M 차종 SP7 *)
    S365_M_차종_SP8 AT %MW10150.7 : BOOL; (* S365 M 차종 SP8 *)
    S365_M_차종_SP9 AT %MW10150.15 : BOOL; (* S365 M 차종 SP9 *)
    S365_M_차종_공대차 AT %MW10150.12 : BOOL; (* S365 M 차종 공대차 *)
    S365_M_차종_공차 AT %MW10150.10 : BOOL; (* S365 M 차종 공차 *)
    S365_M_차종_불량대차 AT %MW10150.13 : BOOL; (* S365 M 차종 불량대차 *)
    S365_M_차종_불량차 AT %MW10150.11 : BOOL; (* S365 M 차종 불량차 *)
    S365_M_차종_비축 AT %MW10150.8 : BOOL; (* S365 M 차종 비축 *)
    S365_M_차종_취출대차 AT %MW10150.14 : BOOL; (* S365 M 차종 취출대차 *)
    S365_M_총괄_CP_이상 AT %MW2509.7 : BOOL; (* S365 CP OFF 이상 *)
    S365_M_총괄_CT_이상 AT %MW2510.4 : BOOL; (* S365   TACK TIME 이상 *)
    S365_M_총괄_EOCR_이상 AT %MW2509.8 : BOOL; (* S365_M_총괄_EOCR_이상 *)
    S365_M_총괄_INV_이상 AT %MW2509.9 : BOOL; (* S365_M_총괄_INV_이상 *)
    S365_M_총괄_LS_이상 AT %MW2509.15 : BOOL; (* S365 LS 이상 *)
    S365_M_총괄_MATCH_이상 AT %MW2510.0 : BOOL; (* S365 매트SW 이상 *)
    S365_M_총괄_MC_이상 AT %MW2509.13 : BOOL; (* S365_M_총괄_MC_이상 *)
    S365_M_총괄_MOTOR_이상 AT %MW2510.3 : BOOL; (* S365_M_총괄_MOTOR_이상 *)
    S365_M_총괄_NFB_이상 AT %MW2509.11 : BOOL; (* S365_M_총괄_NFB_이상 *)
    S365_M_총괄_ROBOT_이상 AT %MW2510.1 : BOOL; (* S365 ROBOT 이상 *)
    S365_M_총괄_SAFETY_이상 AT %MW2509.2 : BOOL; (* S365 SAFETY 이상 *)
    S365_M_총괄_SRV_이상 AT %MW2509.10 : BOOL; (* S365_M_총괄_SRV_이상 *)
    S365_M_총괄_공기압_이상 AT %MW2509.3 : BOOL; (* S365 공기압 이상 *)
    S365_M_총괄_비상정지_이상 AT %MW2509.1 : BOOL; (* S365_M_총괄_비상정지_이상 *)
    S365_M_총괄_사양_이상 AT %MW2509.6 : BOOL; (* S365 사양 이상 *)
    S365_M_총괄_오버런_이상 AT %MW2509.12 : BOOL; (* S365_M_총괄_오버런_이상 *)
    S365_M_총괄_용접타점수_이상 AT %MW2510.2 : BOOL; (* S365 용접타점수 이상 *)
    S365_M_총괄_이상 AT %MW2509.0 : BOOL; (* S365_M_총괄_이상 *)
    S365_M_총괄_제품감지_이상 AT %MW2509.4 : BOOL; (* S365 제품감지 이상 *)
    S365_M_총괄_차종_이상 AT %MW2509.5 : BOOL; (* S365 차종 이상 *)
    S365_M_총괄_통신_이상 AT %MW2509.14 : BOOL; (* S365 통신이상 *)
    S365_전진_ON AT %MW2548.1 : BOOL; (* S365_전진_ON *)
    S365_후진_ON AT %MW2548.2 : BOOL; (* S365_후진_ON *)
    S366_HOME AT %MW3048.0 : BOOL; (* S366_HOME *)
    S366_LH_M_NODE_8_10_통신_이상 AT %MW3024.1 : BOOL;
    S366_M_AX_LH_CLP_전진_LS_이상 AT %MW3104.5 : BOOL; (* S366_M_AX_LH_CLP_전진_LS_이상 *)
    S366_M_AX_LH_CLP_전진_보조 AT %MW3104.1 : BOOL; (* S366_M_AX_LH_CLP_전진_보조 *)
    S366_M_AX_LH_CLP_전진단 AT %MW3104.3 : BOOL; (* S366_M_AX_LH_CLP_전진단 *)
    S366_M_AX_LH_CLP_조건 AT %MW3104.0 : BOOL; (* S366_M_AX_LH_CLP_조건 *)
    S366_M_AX_LH_CLP_후진_LS_이상 AT %MW3104.6 : BOOL; (* S366_M_AX_LH_CLP_후진_LS_이상 *)
    S366_M_AX_LH_CLP_후진_보조 AT %MW3104.2 : BOOL; (* S366_M_AX_LH_CLP_후진_보조 *)
    S366_M_AX_LH_CLP_후진단 AT %MW3104.4 : BOOL; (* S366_M_AX_LH_CLP_후진단 *)
    S366_M_AX_RH_CLP_전진_LS_이상 AT %MW3112.5 : BOOL; (* S366_M_AX_RH_CLP_전진_LS_이상 *)
    S366_M_AX_RH_CLP_전진_보조 AT %MW3112.1 : BOOL; (* S366_M_AX_RH_CLP_전진_보조 *)
    S366_M_AX_RH_CLP_전진단 AT %MW3112.3 : BOOL; (* S366_M_AX_RH_CLP_전진단 *)
    S366_M_AX_RH_CLP_조건 AT %MW3112.0 : BOOL; (* S366_M_AX_RH_CLP_조건 *)
    S366_M_AX_RH_CLP_후진_LS_이상 AT %MW3112.6 : BOOL; (* S366_M_AX_RH_CLP_후진_LS_이상 *)
    S366_M_AX_RH_CLP_후진_보조 AT %MW3112.2 : BOOL; (* S366_M_AX_RH_CLP_후진_보조 *)
    S366_M_AX_RH_CLP_후진단 AT %MW3112.4 : BOOL; (* S366_M_AX_RH_CLP_후진단 *)
    S366_M_BYPASS_보조 AT %MW3003.15 : BOOL; (* S366 M BYPASS 보조 *)
    S366_M_CP_OFF AT %MW3017.0 : BOOL;
    S366_M_CTIME_OVER_ALRAM AT %MW3007.14 : BOOL; (* S366_M_CTIME_OVER_ALRAM *)
    S366_M_CTIME_OVER_MUTE AT %MW3007.13 : BOOL; (* S366_M_CTIME_OVER_MUTE *)
    S366_M_DATA_삭제_PLS AT %MW9014.0 : BOOL; (* S366 M DATA 삭제 PLS *)
    S366_M_DATA_삭제_SIGN AT %MW9014.1 : BOOL; (* S366 M DATA 삭제 SIGN *)
    S366_M_DATA_삭제_완료 AT %MW9014.2 : BOOL; (* S366 M DATA 삭제 완료 *)
    S366_M_LC_정상 AT %MW3007.5 : BOOL; (* S366_M_LC_정상 *)
    S366_M_LH_CB_OFF AT %MW3021.2 : BOOL;
    S366_M_LH_CP_OFF AT %MW3017.2 : BOOL; (* S366_M_LH_CP_OFF *)
    S366_M_LH_INV_이상 AT %MW3019.0 : BOOL; (* S366_M_LH_INV_이상 *)
    S366_M_LH_MAIN_BAR_이상 AT %MW3012.0 : BOOL; (* S366_M_LH_MAIN_BAR_이상 *)
    S366_M_LH_MC_이상 AT %MW3023.0 : BOOL; (* S366_M_LH_MC_이상 *)
    S366_M_LH_NFB_OFF AT %MW3021.0 : BOOL; (* S366_M_LH_NFB_OFF *)
    S366_M_LH_STEP_MOVE_리셋_PLS AT %MW3101.14 : BOOL; (* S366_M_LH_STEP_MOVE_리셋_PLS *)
    S366_M_LH_TURN_1_포지션단 AT %MW3101.3 : BOOL; (* S366_M_LH_TURN_1_포지션단 *)
    S366_M_LH_TURN_2_포지션단 AT %MW3101.4 : BOOL; (* S366_M_LH_TURN_2_포지션단 *)
    S366_M_LH_TURN_3_포지션단 AT %MW3101.5 : BOOL; (* S366_M_LH_TURN_3_포지션단 *)
    S366_M_LH_TURN_4_포지션단 AT %MW3101.6 : BOOL; (* S366_M_LH_TURN_4_포지션단 *)
    S366_M_LH_TURN_LS_이상 AT %MW3101.7 : BOOL; (* S366_M_LH_TURN_LS_이상 *)
    S366_M_LH_TURN_MOVE_완료 AT %MW3101.8 : BOOL; (* S366_M_LH_TURN_MOVE_완료 *)
    S366_M_LH_TURN_수동_STEP_전진_보조 AT %MW3101.11 : BOOL; (* S366_M_LH_TURN_수동_STEP_전진_보조 *)
    S366_M_LH_TURN_수동_STEP_후진_보조 AT %MW3101.12 : BOOL; (* S366_M_LH_TURN_수동_STEP_후진_보조 *)
    S366_M_LH_TURN_수동_전진_보조 AT %MW3101.9 : BOOL; (* S366_M_LH_TURN_수동_전진_보조 *)
    S366_M_LH_TURN_수동_후진_보조 AT %MW3101.10 : BOOL; (* S366_M_LH_TURN_수동_후진_보조 *)
    S366_M_LH_TURN_전진_보조 AT %MW3101.1 : BOOL; (* S366_M_LH_TURN_전진_보조 *)
    S366_M_LH_TURN_조건 AT %MW3101.0 : BOOL; (* S366_M_LH_TURN_조건 *)
    S366_M_LH_TURN_후진_보조 AT %MW3101.2 : BOOL; (* S366_M_LH_TURN_후진_보조 *)
    S366_M_LH_공기압_이상 AT %MW3013.0 : BOOL; (* S366_M_LH_공기압_이상 *)
    S366_M_LH_자동_MOVE_리셋_PLS AT %MW3101.13 : BOOL; (* S366_M_LH_자동_MOVE_리셋_PLS *)
    S366_M_MAT_정상 AT %MW3007.6 : BOOL; (* S366_M_MAT_정상 *)
    S366_M_NODE_6_10_통신_이상 AT %MW3024.0 : BOOL;
    S366_M_OP_ESTOP_NORMAL AT %MW3007.1 : BOOL; (* S366_M_OP_ESTOP_NORMAL *)
    S366_M_R361_1_DATA_전송_MEMO AT %MW9014.8 : BOOL; (* S366 M R361 1 DATA 전송 MEMO *)
    S366_M_R361_1_DATA_전송_PLS AT %MW9014.9 : BOOL; (* S366 M R361 1 DATA 전송 PLS *)
    S366_M_R361_1_DATA_전송_SIGN AT %MW9014.10 : BOOL; (* S366 M R361 1 DATA 전송 SIGN *)
    S366_M_R361_1_DATA_전송_완료 AT %MW9014.11 : BOOL; (* S366 M R361 1 DATA 전송 완료 *)
    S366_M_R361_1_ROOF_로딩완료 AT %MW3001.2 : BOOL;
    S366_M_R361_1_동일차종_OK AT %MW3005.8 : BOOL;
    S366_M_R361_1_언로딩완료 AT %MW3001.4 : BOOL;
    S366_M_R361_1_차종매칭_조건 AT %MW3005.0 : BOOL;
    S366_M_R363_2_RAIL_로딩완료 AT %MW3001.1 : BOOL;
    S366_M_R366_1_용접가능 AT %MW3004.10 : BOOL;
    S366_M_R366_1_용접완료 AT %MW3001.3 : BOOL;
    S366_M_RAIL_로딩가능 AT %MW3004.8 : BOOL;
    S366_M_RH_CB_OFF AT %MW3021.3 : BOOL;
    S366_M_RH_CP_OFF AT %MW3017.3 : BOOL; (* S366_M_RH_CP_OFF *)
    S366_M_RH_INV_이상 AT %MW3019.1 : BOOL; (* S366_M_RH_INV_이상 *)
    S366_M_RH_MAIN_BAR_이상 AT %MW3012.1 : BOOL; (* S366_M_RH_MAIN_BAR_이상 *)
    S366_M_RH_MC_이상 AT %MW3023.1 : BOOL; (* S366_M_RH_MC_이상 *)
    S366_M_RH_NFB_OFF AT %MW3021.1 : BOOL; (* S366_M_RH_NFB_OFF *)
    S366_M_RH_STEP_MOVE_리셋_PLS AT %MW3109.14 : BOOL; (* S366_M_RH_STEP_MOVE_리셋_PLS *)
    S366_M_RH_TURN_1_포지션단 AT %MW3109.3 : BOOL; (* S366_M_RH_TURN_1_포지션단 *)
    S366_M_RH_TURN_2_포지션단 AT %MW3109.4 : BOOL; (* S366_M_RH_TURN_2_포지션단 *)
    S366_M_RH_TURN_3_포지션단 AT %MW3109.5 : BOOL; (* S366_M_RH_TURN_3_포지션단 *)
    S366_M_RH_TURN_4_포지션단 AT %MW3109.6 : BOOL; (* S366_M_RH_TURN_4_포지션단 *)
    S366_M_RH_TURN_LS_이상 AT %MW3109.7 : BOOL; (* S366_M_RH_TURN_LS_이상 *)
    S366_M_RH_TURN_MOVE_완료 AT %MW3109.8 : BOOL; (* S366_M_RH_TURN_MOVE_완료 *)
    S366_M_RH_TURN_수동_STEP_전진_보조 AT %MW3109.11 : BOOL; (* S366_M_RH_TURN_수동_STEP_전진_보조 *)
    S366_M_RH_TURN_수동_STEP_후진_보조 AT %MW3109.12 : BOOL; (* S366_M_RH_TURN_수동_STEP_후진_보조 *)
    S366_M_RH_TURN_수동_전진_보조 AT %MW3109.9 : BOOL; (* S366_M_RH_TURN_수동_전진_보조 *)
    S366_M_RH_TURN_수동_후진_보조 AT %MW3109.10 : BOOL; (* S366_M_RH_TURN_수동_후진_보조 *)
    S366_M_RH_TURN_전진_보조 AT %MW3109.1 : BOOL; (* S366_M_RH_TURN_전진_보조 *)
    S366_M_RH_TURN_조건 AT %MW3109.0 : BOOL; (* S366_M_RH_TURN_조건 *)
    S366_M_RH_TURN_후진_보조 AT %MW3109.2 : BOOL; (* S366_M_RH_TURN_후진_보조 *)
    S366_M_RH_공기압_이상 AT %MW3013.1 : BOOL; (* S366_M_RH_공기압_이상 *)
    S366_M_RH_자동_MOVE_리셋_PLS AT %MW3109.13 : BOOL; (* S366_M_RH_자동_MOVE_리셋_PLS *)
    S366_M_ROOF_로딩가능 AT %MW3004.9 : BOOL;
    S366_M_SAFETY_불간섭 AT %MW3004.4 : BOOL; (* S366_M_SAFETY_불간섭 *)
    S366_M_SEMI_자동모드 AT %MW3000.2 : BOOL; (* S366_M_SEMI_자동모드 *)
    S366_M_SEQ AT %MW10160 : WORD; (* S366 M SEQ *)
    S366_M_TURN_LOCK_전진_LS_이상 AT %MW3100.5 : BOOL; (* S366_M_TURN_LOCK_전진_LS_이상 *)
    S366_M_TURN_LOCK_전진_보조 AT %MW3100.1 : BOOL; (* S366_M_TURN_LOCK_전진_보조 *)
    S366_M_TURN_LOCK_전진단 AT %MW3100.3 : BOOL; (* S366_M_TURN_LOCK_전진단 *)
    S366_M_TURN_LOCK_조건 AT %MW3100.0 : BOOL; (* S366_M_TURN_LOCK_조건 *)
    S366_M_TURN_LOCK_후진_LS_이상 AT %MW3100.6 : BOOL; (* S366_M_TURN_LOCK_후진_LS_이상 *)
    S366_M_TURN_LOCK_후진_보조 AT %MW3100.2 : BOOL; (* S366_M_TURN_LOCK_후진_보조 *)
    S366_M_TURN_LOCK_후진단 AT %MW3100.4 : BOOL; (* S366_M_TURN_LOCK_후진단 *)
    S366_M_VIN_NO_1_2 AT %MW10171 : WORD; (* S366 M VIN NO 1 2 *)
    S366_M_VIN_NO_3_4 AT %MW10172 : WORD; (* S366 M VIN NO 3 4 *)
    S366_M_VIN_NO_5_6 AT %MW10173 : WORD; (* S366 M VIN NO 5 6 *)
    S366_M_VIN_NO_7_8 AT %MW10174 : WORD; (* S366 M VIN NO 7 8 *)
    S366_M_VIN_NO_9_10 AT %MW10175 : WORD; (* S366 M VIN NO 9 10 *)
    S366_M_공정_AX_FRT_PNL_제품감지_이상 AT %MW3014.4 : BOOL;
    S366_M_공정_AX_RAIL_제품감지_이상 AT %MW3014.3 : BOOL;
    S366_M_공정_AX_RR_PNL_제품감지_이상 AT %MW3014.5 : BOOL;
    S366_M_공정_AX_공용_제품감지_이상 AT %MW3014.0 : BOOL;
    S366_M_공정_AX_썬루프_제품감지_이상 AT %MW3014.2 : BOOL;
    S366_M_공정_AX_일반루프_제품감지_이상 AT %MW3014.1 : BOOL;
    S366_M_공정_FRT_PNL_제품감지_무 AT %MW3002.13 : BOOL;
    S366_M_공정_FRT_PNL_제품감지_유 AT %MW3002.12 : BOOL;
    S366_M_공정_RAIL_제품감지_무 AT %MW3001.15 : BOOL;
    S366_M_공정_RAIL_제품감지_유 AT %MW3001.14 : BOOL;
    S366_M_공정_RR_PNL_제품감지_무 AT %MW3002.15 : BOOL;
    S366_M_공정_RR_PNL_제품감지_유 AT %MW3002.14 : BOOL;
    S366_M_공정_SAFETY_NORMAL AT %MW3007.7 : BOOL; (* S366_M_공정_SAFETY_NORMAL *)
    S366_M_공정_공용_제품감지_무 AT %MW3001.9 : BOOL;
    S366_M_공정_공용_제품감지_유 AT %MW3001.8 : BOOL;
    S366_M_공정_불간섭 AT %MW3004.1 : BOOL; (* S366_M_공정_불간섭 *)
    S366_M_공정_썬루프_제품감지_무 AT %MW3001.13 : BOOL;
    S366_M_공정_썬루프_제품감지_유 AT %MW3001.12 : BOOL;
    S366_M_공정_원위치 AT %MW3004.0 : BOOL; (* S366_M_공정_원위치 *)
    S366_M_공정_일반루프_제품감지_무 AT %MW3001.11 : BOOL;
    S366_M_공정_일반루프_제품감지_유 AT %MW3001.10 : BOOL;
    S366_M_공정_제품감지_무 AT %MW3001.7 : BOOL; (* S366_M_공정_제품감지_무 *)
    S366_M_공정_제품감지_유 AT %MW3001.6 : BOOL; (* S366_M_공정_제품감지_유 *)
    S366_M_공정_차종_AX AT %MW3002.3 : BOOL; (* S366_M_공정_차종_AX *)
    S366_M_공정_차종_무 AT %MW3002.1 : BOOL; (* S366_M_공정_차종_무 *)
    S366_M_공정_차종_유 AT %MW3002.0 : BOOL; (* S366_M_공정_차종_유 *)
    S366_M_동작_선택_1 AT %MW3040.0 : BOOL; (* S366_M_동작_선택_1 *)
    S366_M_동작_선택_10 AT %MW3040.9 : BOOL; (* S366_M_동작_선택_10 *)
    S366_M_동작_선택_11 AT %MW3040.10 : BOOL; (* S366_M_동작_선택_11 *)
    S366_M_동작_선택_12 AT %MW3040.11 : BOOL; (* S366_M_동작_선택_12 *)
    S366_M_동작_선택_13 AT %MW3040.12 : BOOL; (* S366_M_동작_선택_13 *)
    S366_M_동작_선택_14 AT %MW3040.13 : BOOL; (* S366_M_동작_선택_14 *)
    S366_M_동작_선택_15 AT %MW3040.14 : BOOL; (* S366_M_동작_선택_15 *)
    S366_M_동작_선택_16 AT %MW3040.15 : BOOL; (* S366_M_동작_선택_16 *)
    S366_M_동작_선택_17 AT %MW3041.0 : BOOL; (* S366_M_동작_선택_17 *)
    S366_M_동작_선택_18 AT %MW3041.1 : BOOL; (* S366_M_동작_선택_18 *)
    S366_M_동작_선택_19 AT %MW3041.2 : BOOL; (* S366_M_동작_선택_19 *)
    S366_M_동작_선택_2 AT %MW3040.1 : BOOL; (* S366_M_동작_선택_2 *)
    S366_M_동작_선택_20 AT %MW3041.3 : BOOL; (* S366_M_동작_선택_20 *)
    S366_M_동작_선택_21 AT %MW3041.4 : BOOL; (* S366_M_동작_선택_21 *)
    S366_M_동작_선택_22 AT %MW3041.5 : BOOL; (* S366_M_동작_선택_22 *)
    S366_M_동작_선택_23 AT %MW3041.6 : BOOL; (* S366_M_동작_선택_23 *)
    S366_M_동작_선택_24 AT %MW3041.7 : BOOL; (* S366_M_동작_선택_24 *)
    S366_M_동작_선택_25 AT %MW3041.8 : BOOL; (* S366_M_동작_선택_25 *)
    S366_M_동작_선택_26 AT %MW3041.9 : BOOL; (* S366_M_동작_선택_26 *)
    S366_M_동작_선택_27 AT %MW3041.10 : BOOL; (* S366_M_동작_선택_27 *)
    S366_M_동작_선택_28 AT %MW3041.11 : BOOL; (* S366_M_동작_선택_28 *)
    S366_M_동작_선택_29 AT %MW3041.12 : BOOL; (* S366_M_동작_선택_29 *)
    S366_M_동작_선택_3 AT %MW3040.2 : BOOL; (* S366_M_동작_선택_3 *)
    S366_M_동작_선택_30 AT %MW3041.13 : BOOL; (* S366_M_동작_선택_30 *)
    S366_M_동작_선택_31 AT %MW3041.14 : BOOL; (* S366_M_동작_선택_31 *)
    S366_M_동작_선택_32 AT %MW3041.15 : BOOL; (* S366_M_동작_선택_32 *)
    S366_M_동작_선택_4 AT %MW3040.3 : BOOL; (* S366_M_동작_선택_4 *)
    S366_M_동작_선택_5 AT %MW3040.4 : BOOL; (* S366_M_동작_선택_5 *)
    S366_M_동작_선택_6 AT %MW3040.5 : BOOL; (* S366_M_동작_선택_6 *)
    S366_M_동작_선택_7 AT %MW3040.6 : BOOL; (* S366_M_동작_선택_7 *)
    S366_M_동작_선택_8 AT %MW3040.7 : BOOL; (* S366_M_동작_선택_8 *)
    S366_M_동작_선택_9 AT %MW3040.8 : BOOL; (* S366_M_동작_선택_9 *)
    S366_M_부저_정지_보조 AT %MW3000.11 : BOOL; (* S366_M_부저_정지_보조 *)
    S366_M_수동모드 AT %MW3000.3 : BOOL; (* S366 선택 수동모드 *)
    S366_M_썬루프_사양_이상 AT %MW3016.1 : BOOL;
    S366_M_운전준비_ON AT %MW3000.0 : BOOL; (* S366 운전준비 ON *)
    S366_M_이상_리셋_보조 AT %MW3000.10 : BOOL; (* S366_M_이상_리셋_보조 *)
    S366_M_일반루프_사양_이상 AT %MW3016.0 : BOOL;
    S366_M_자동_START AT %MW3000.5 : BOOL; (* S366 자동운전중 *)
    S366_M_자동_운전중 AT %MW3000.4 : BOOL; (* S366 자동운전중 *)
    S366_M_자동모드 AT %MW3000.1 : BOOL; (* S366 선택 자동모드 *)
    S366_M_작업_완료 AT %MW3001.0 : BOOL; (* S366_M_작업_완료 *)
    S366_M_작업완료_SET_PLS AT %MW3000.8 : BOOL; (* S366 M 작업완료 SET PLS *)
    S366_M_작업완료_리셋_PLS AT %MW3000.9 : BOOL; (* S366 M 작업완료 리셋 PLS *)
    S366_M_전체_용접완료 AT %MW3006.0 : BOOL;
    S366_M_차종1_AX AT %MW10161.0 : BOOL; (* S366 M 차종1 AX *)
    S366_M_차종1_B AT %MW10161.1 : BOOL; (* S366 M 차종1 B *)
    S366_M_차종1_C AT %MW10161.2 : BOOL; (* S366 M 차종1 C *)
    S366_M_차종1_D AT %MW10161.3 : BOOL; (* S366 M 차종1 D *)
    S366_M_차종1_E AT %MW10161.4 : BOOL; (* S366 M 차종1 E *)
    S366_M_차종1_F AT %MW10161.5 : BOOL; (* S366 M 차종1 F *)
    S366_M_차종1_G AT %MW10161.6 : BOOL; (* S366 M 차종1 G *)
    S366_M_차종1_H AT %MW10161.7 : BOOL; (* S366 M 차종1 H *)
    S366_M_차종2_3DR AT %MW10161.8 : BOOL; (* S366 M 차종2 3DR *)
    S366_M_차종2_4DR AT %MW10161.9 : BOOL; (* S366 M 차종2 4DR *)
    S366_M_차종2_5DR AT %MW10161.10 : BOOL; (* S366 M 차종2 5DR *)
    S366_M_차종2_SP1 AT %MW10161.12 : BOOL; (* S366 M 차종2 SP1 *)
    S366_M_차종2_SP2 AT %MW10161.13 : BOOL; (* S366 M 차종2 SP2 *)
    S366_M_차종2_WGN AT %MW10161.11 : BOOL; (* S366 M 차종2 WGN *)
    S366_M_차종3_LHD AT %MW10161.14 : BOOL; (* S366 M 차종3 LHD *)
    S366_M_차종3_RHD AT %MW10161.15 : BOOL; (* S366 M 차종3 RHD *)
    S366_M_차종4_EEC AT %MW10162.3 : BOOL; (* S366 M 차종4 EEC *)
    S366_M_차종4_SP1 AT %MW10162.8 : BOOL; (* S366 M 차종4 SP1 *)
    S366_M_차종4_SP2 AT %MW10162.9 : BOOL; (* S366 M 차종4 SP2 *)
    S366_M_차종4_SP3 AT %MW10162.11 : BOOL; (* S366 M 차종4 SP3 *)
    S366_M_차종4_SP4 AT %MW10162.12 : BOOL; (* S366 M 차종4 SP4 *)
    S366_M_차종4_SP5 AT %MW10162.13 : BOOL; (* S366 M 차종4 SP5 *)
    S366_M_차종4_SP6 AT %MW10162.14 : BOOL; (* S366 M 차종4 SP6 *)
    S366_M_차종4_SP7 AT %MW10162.15 : BOOL; (* S366 M 차종4 SP7 *)
    S366_M_차종4_내수 AT %MW10162.0 : BOOL; (* S366 M 차종4 내수 *)
    S366_M_차종4_러시아 AT %MW10162.10 : BOOL; (* S366 M 차종4 러시아 *)
    S366_M_차종4_북미 AT %MW10162.2 : BOOL; (* S366 M 차종4 북미 *)
    S366_M_차종4_브라질 AT %MW10162.7 : BOOL; (* S366 M 차종4 브라질 *)
    S366_M_차종4_수출 AT %MW10162.1 : BOOL; (* S366 M 차종4 수출 *)
    S366_M_차종4_중국 AT %MW10162.6 : BOOL; (* S366 M 차종4 중국 *)
    S366_M_차종4_중동 AT %MW10162.5 : BOOL; (* S366 M 차종4 중동 *)
    S366_M_차종4_호주 AT %MW10162.4 : BOOL; (* S366 M 차종4 호주 *)
    S366_M_차종5_AT AT %MW10163.1 : BOOL; (* S366 M 차종5 AT *)
    S366_M_차종5_MT AT %MW10163.0 : BOOL; (* S366 M 차종5 MT *)
    S366_M_차종5_SP1 AT %MW10163.2 : BOOL; (* S366 M 차종5 SP1 *)
    S366_M_차종6_DSROOF AT %MW10163.6 : BOOL; (* S366 M 차종6 DSROOF *)
    S366_M_차종6_SP1 AT %MW10163.7 : BOOL; (* S366 M 차종6 SP1 *)
    S366_M_차종6_썬루프 AT %MW10163.4 : BOOL; (* S366 M 차종6 썬루프 *)
    S366_M_차종6_일반루프 AT %MW10163.3 : BOOL; (* S366 M 차종6 일반루프 *)
    S366_M_차종6_파노라마루프 AT %MW10163.5 : BOOL; (* S366 M 차종6 파노라마루프 *)
    S366_M_차종7_DSL AT %MW10163.9 : BOOL; (* S366 M 차종7 DSL *)
    S366_M_차종7_GSL AT %MW10163.8 : BOOL; (* S366 M 차종7 GSL *)
    S366_M_차종7_SP1 AT %MW10163.10 : BOOL; (* S366 M 차종7 SP1 *)
    S366_M_차종7_SP2 AT %MW10163.11 : BOOL; (* S366 M 차종7 SP2 *)
    S366_M_차종7_SP3 AT %MW10163.12 : BOOL; (* S366 M 차종7 SP3 *)
    S366_M_차종7_SP4 AT %MW10163.13 : BOOL; (* S366 M 차종7 SP4 *)
    S366_M_차종7_SP5 AT %MW10163.14 : BOOL; (* S366 M 차종7 SP5 *)
    S366_M_차종7_SP6 AT %MW10163.15 : BOOL; (* S366 M 차종7 SP6 *)
    S366_M_차종8_2WD AT %MW10164.0 : BOOL; (* S366 M 차종8 2WD *)
    S366_M_차종8_4WD AT %MW10164.1 : BOOL; (* S366 M 차종8 4WD *)
    S366_M_차종8_SP1 AT %MW10164.2 : BOOL; (* S366 M 차종8 SP1 *)
    S366_M_차종9_MPI AT %MW10164.3 : BOOL; (* S366 M 차종9 MPI *)
    S366_M_차종9_SP1 AT %MW10164.5 : BOOL; (* S366 M 차종9 SP1 *)
    S366_M_차종9_SP10 AT %MW10164.14 : BOOL; (* S366 M 차종9 SP10 *)
    S366_M_차종9_SP11 AT %MW10164.15 : BOOL; (* S366 M 차종9 SP11 *)
    S366_M_차종9_SP2 AT %MW10164.6 : BOOL; (* S366 M 차종9 SP2 *)
    S366_M_차종9_SP3 AT %MW10164.7 : BOOL; (* S366 M 차종9 SP3 *)
    S366_M_차종9_SP4 AT %MW10164.8 : BOOL; (* S366 M 차종9 SP4 *)
    S366_M_차종9_SP5 AT %MW10164.9 : BOOL; (* S366 M 차종9 SP5 *)
    S366_M_차종9_SP6 AT %MW10164.10 : BOOL; (* S366 M 차종9 SP6 *)
    S366_M_차종9_SP7 AT %MW10164.11 : BOOL; (* S366 M 차종9 SP7 *)
    S366_M_차종9_SP8 AT %MW10164.12 : BOOL; (* S366 M 차종9 SP8 *)
    S366_M_차종9_SP9 AT %MW10164.13 : BOOL; (* S366 M 차종9 SP9 *)
    S366_M_차종9_T_GDI AT %MW10164.4 : BOOL; (* S366 M 차종9 T GDI *)
    S366_M_차종_AS AT %MW10170.9 : BOOL; (* S366 M 차종 AS *)
    S366_M_차종_OPT1_R_RACK_무 AT %MW10165.3 : BOOL; (* S366 M 차종 OPT1 R RACK 무 *)
    S366_M_차종_OPT1_R_RACK_유 AT %MW10165.2 : BOOL; (* S366 M 차종 OPT1 R RACK 유 *)
    S366_M_차종_OPT1_SP1 AT %MW10165.10 : BOOL; (* S366 M 차종 OPT1 SP1 *)
    S366_M_차종_OPT1_SP2 AT %MW10165.11 : BOOL; (* S366 M 차종 OPT1 SP2 *)
    S366_M_차종_OPT1_SP3 AT %MW10165.12 : BOOL; (* S366 M 차종 OPT1 SP3 *)
    S366_M_차종_OPT1_SP4 AT %MW10165.13 : BOOL; (* S366 M 차종 OPT1 SP4 *)
    S366_M_차종_OPT1_SP5 AT %MW10165.14 : BOOL; (* S366 M 차종 OPT1 SP5 *)
    S366_M_차종_OPT1_SP6 AT %MW10165.15 : BOOL; (* S366 M 차종 OPT1 SP6 *)
    S366_M_차종_OPT1_S_REP_EATER_무 AT %MW10165.7 : BOOL; (* S366 M 차종 OPT1 S REP EATER 무 *)
    S366_M_차종_OPT1_S_REP_EATER_유 AT %MW10165.6 : BOOL; (* S366 M 차종 OPT1 S REP EATER 유 *)
    S366_M_차종_OPT1_VAN_무 AT %MW10165.9 : BOOL; (* S366 M 차종 OPT1 VAN 무 *)
    S366_M_차종_OPT1_VAN_유 AT %MW10165.8 : BOOL; (* S366 M 차종 OPT1 VAN 유 *)
    S366_M_차종_OPT1_슬라이딩_무 AT %MW10165.1 : BOOL; (* S366 M 차종 OPT1 슬라이딩 무 *)
    S366_M_차종_OPT1_슬라이딩_유 AT %MW10165.0 : BOOL; (* S366 M 차종 OPT1 슬라이딩 유 *)
    S366_M_차종_OPT1_폴딩_무 AT %MW10165.5 : BOOL; (* S366 M 차종 OPT1 폴딩 무 *)
    S366_M_차종_OPT1_폴딩_유 AT %MW10165.4 : BOOL; (* S366 M 차종 OPT1 폴딩 유 *)
    S366_M_차종_OPT2_SP_WORD1 AT %MW10166 : WORD; (* S366 M 차종 OPT2 SP WORD1 *)
    S366_M_차종_OPT3_SP_WORD2 AT %MW10167 : WORD; (* S366 M 차종 OPT3 SP WORD2 *)
    S366_M_차종_OPT4_SP_WORD3 AT %MW10168 : WORD; (* S366 M 차종 OPT4 SP WORD3 *)
    S366_M_차종_OPT5_SP_WORD4 AT %MW10169 : WORD; (* S366 M 차종 OPT5 SP WORD4 *)
    S366_M_차종_SP1 AT %MW10170.0 : BOOL; (* S366 M 차종 SP1 *)
    S366_M_차종_SP2 AT %MW10170.1 : BOOL; (* S366 M 차종 SP2 *)
    S366_M_차종_SP3 AT %MW10170.2 : BOOL; (* S366 M 차종 SP3 *)
    S366_M_차종_SP4 AT %MW10170.3 : BOOL; (* S366 M 차종 SP4 *)
    S366_M_차종_SP5 AT %MW10170.4 : BOOL; (* S366 M 차종 SP5 *)
    S366_M_차종_SP6 AT %MW10170.5 : BOOL; (* S366 M 차종 SP6 *)
    S366_M_차종_SP7 AT %MW10170.6 : BOOL; (* S366 M 차종 SP7 *)
    S366_M_차종_SP8 AT %MW10170.7 : BOOL; (* S366 M 차종 SP8 *)
    S366_M_차종_SP9 AT %MW10170.15 : BOOL; (* S366 M 차종 SP9 *)
    S366_M_차종_공대차 AT %MW10170.12 : BOOL; (* S366 M 차종 공대차 *)
    S366_M_차종_공차 AT %MW10170.10 : BOOL; (* S366 M 차종 공차 *)
    S366_M_차종_불량대차 AT %MW10170.13 : BOOL; (* S366 M 차종 불량대차 *)
    S366_M_차종_불량차 AT %MW10170.11 : BOOL; (* S366 M 차종 불량차 *)
    S366_M_차종_비축 AT %MW10170.8 : BOOL; (* S366 M 차종 비축 *)
    S366_M_차종_취출대차 AT %MW10170.14 : BOOL; (* S366 M 차종 취출대차 *)
    S366_M_총괄_CP_이상 AT %MW3009.7 : BOOL; (* S366 CP OFF 이상 *)
    S366_M_총괄_CT_이상 AT %MW3010.4 : BOOL; (* S366   TACK TIME 이상 *)
    S366_M_총괄_EOCR_이상 AT %MW3009.8 : BOOL; (* S366_M_총괄_EOCR_이상 *)
    S366_M_총괄_INV_이상 AT %MW3009.9 : BOOL; (* S366 인버터 이상 *)
    S366_M_총괄_LS_이상 AT %MW3009.15 : BOOL; (* S366 LS 이상 *)
    S366_M_총괄_MATCH_이상 AT %MW3010.0 : BOOL; (* S366 매트SW 이상 *)
    S366_M_총괄_MC_이상 AT %MW3009.13 : BOOL; (* S366 MC 이상 *)
    S366_M_총괄_MOTOR_이상 AT %MW3010.3 : BOOL; (* S366 MOTOR 이상 *)
    S366_M_총괄_NFB_이상 AT %MW3009.11 : BOOL; (* S366 NFB 이상 *)
    S366_M_총괄_ROBOT_이상 AT %MW3010.1 : BOOL; (* S366 ROBOT 이상 *)
    S366_M_총괄_SAFETY_이상 AT %MW3009.2 : BOOL; (* S366_M_총괄_SAFETY_이상 *)
    S366_M_총괄_SRV_이상 AT %MW3009.10 : BOOL; (* S366_M_총괄_SRV_이상 *)
    S366_M_총괄_공기압_이상 AT %MW3009.3 : BOOL; (* S366 공기압 이상 *)
    S366_M_총괄_비상정지_이상 AT %MW3009.1 : BOOL; (* S366_M_총괄_비상정지_이상 *)
    S366_M_총괄_사양_이상 AT %MW3009.6 : BOOL; (* S366 사양 이상 *)
    S366_M_총괄_오버런_이상 AT %MW3009.12 : BOOL; (* S366 OVER RUN 이상 *)
    S366_M_총괄_용접타점수_이상 AT %MW3010.2 : BOOL; (* S366 용접타점수 이상 *)
    S366_M_총괄_이상 AT %MW3009.0 : BOOL; (* S366_M_총괄_이상 *)
    S366_M_총괄_제품감지_이상 AT %MW3009.4 : BOOL; (* S366 제품감지 이상 *)
    S366_M_총괄_차종_이상 AT %MW3009.5 : BOOL; (* S366 차종 이상 *)
    S366_M_총괄_통신_이상 AT %MW3009.14 : BOOL; (* S366 통신이상 *)
    S366_RH_M_NODE_8_20_통신_이상 AT %MW3024.2 : BOOL;
    S366_전진_ON AT %MW3048.1 : BOOL; (* S366_전진_ON *)
    S366_후진_ON AT %MW3048.2 : BOOL; (* S366_후진_ON *)
    S367_HOME AT %MW3548.0 : BOOL; (* S367_HOME *)
    S367_LH_M_NODE_6_21_통신_이상 AT %MW3524.0 : BOOL;
    S367_M_369_1_언로딩가능 AT %MW3504.10 : BOOL;
    S367_M_BYPASS_보조 AT %MW3503.15 : BOOL; (* S367 M BYPASS 보조 *)
    S367_M_CTIME_OVER_ALRAM AT %MW3507.14 : BOOL; (* S367_M_CTIME_OVER_ALRAM *)
    S367_M_CTIME_OVER_MUTE AT %MW3507.13 : BOOL; (* S367_M_CTIME_OVER_MUTE *)
    S367_M_DATA_삭제_PLS AT %MW9015.0 : BOOL; (* S367 M DATA 삭제 PLS *)
    S367_M_DATA_삭제_SIGN AT %MW9015.1 : BOOL; (* S367 M DATA 삭제 SIGN *)
    S367_M_DATA_삭제_완료 AT %MW9015.2 : BOOL; (* S367 M DATA 삭제 완료 *)
    S367_M_LC_정상 AT %MW3507.5 : BOOL; (* S367_M_LC_정상 *)
    S367_M_LH_AX_CLAMP_전진_LS_이상 AT %MW3602.5 : BOOL; (* S367_M_LH_AX_CLAMP_전진_LS_이상 *)
    S367_M_LH_AX_CLAMP_전진_보조 AT %MW3602.1 : BOOL; (* S367_M_LH_AX_CLAMP_전진_보조 *)
    S367_M_LH_AX_CLAMP_전진단 AT %MW3602.3 : BOOL; (* S367_M_LH_AX_CLAMP_전진단 *)
    S367_M_LH_AX_CLAMP_조건 AT %MW3602.0 : BOOL; (* S367_M_LH_AX_CLAMP_조건 *)
    S367_M_LH_AX_CLAMP_후진_LS_이상 AT %MW3602.6 : BOOL; (* S367_M_LH_AX_CLAMP_후진_LS_이상 *)
    S367_M_LH_AX_CLAMP_후진_보조 AT %MW3602.2 : BOOL; (* S367_M_LH_AX_CLAMP_후진_보조 *)
    S367_M_LH_AX_CLAMP_후진단 AT %MW3602.4 : BOOL; (* S367_M_LH_AX_CLAMP_후진단 *)
    S367_M_LH_AX_LATCH_전진_LS_이상 AT %MW3600.5 : BOOL; (* S367_M_LH_AX_LATCH_전진_LS_이상 *)
    S367_M_LH_AX_LATCH_전진_보조 AT %MW3600.1 : BOOL; (* S367_M_LH_AX_LATCH_전진_보조 *)
    S367_M_LH_AX_LATCH_전진단 AT %MW3600.3 : BOOL; (* S367_M_LH_AX_LATCH_전진단 *)
    S367_M_LH_AX_LATCH_조건 AT %MW3600.0 : BOOL; (* S367_M_LH_AX_LATCH_조건 *)
    S367_M_LH_AX_LATCH_후진_LS_이상 AT %MW3600.6 : BOOL; (* S367_M_LH_AX_LATCH_후진_LS_이상 *)
    S367_M_LH_AX_LATCH_후진_보조 AT %MW3600.2 : BOOL; (* S367_M_LH_AX_LATCH_후진_보조 *)
    S367_M_LH_AX_LATCH_후진단 AT %MW3600.4 : BOOL; (* S367_M_LH_AX_LATCH_후진단 *)
    S367_M_LH_AX_SR_LAT_전진_LS_이상 AT %MW3601.5 : BOOL; (* S367_M_LH_AX_SR_LAT_전진_LS_이상 *)
    S367_M_LH_AX_SR_LAT_전진_보조 AT %MW3601.1 : BOOL; (* S367_M_LH_AX_SR_LAT_전진_보조 *)
    S367_M_LH_AX_SR_LAT_전진단 AT %MW3601.3 : BOOL; (* S367_M_LH_AX_SR_LAT_전진단 *)
    S367_M_LH_AX_SR_LAT_조건 AT %MW3601.0 : BOOL; (* S367_M_LH_AX_SR_LAT_조건 *)
    S367_M_LH_AX_SR_LAT_후진_LS_이상 AT %MW3601.6 : BOOL; (* S367_M_LH_AX_SR_LAT_후진_LS_이상 *)
    S367_M_LH_AX_SR_LAT_후진_보조 AT %MW3601.2 : BOOL; (* S367_M_LH_AX_SR_LAT_후진_보조 *)
    S367_M_LH_AX_SR_LAT_후진단 AT %MW3601.4 : BOOL; (* S367_M_LH_AX_SR_LAT_후진단 *)
    S367_M_LH_CP_OFF AT %MW3517.0 : BOOL; (* S367_M_LH_CP_OFF *)
    S367_M_LH_공기압_이상 AT %MW3513.0 : BOOL; (* S367_M_LH_공기압_이상 *)
    S367_M_MAT_정상 AT %MW3507.6 : BOOL; (* S367_M_MAT_정상 *)
    S367_M_OP_ESTOP_NORMAL AT %MW3507.1 : BOOL; (* S367_M_OP_ESTOP_NORMAL *)
    S367_M_R361_1_로딩가능 AT %MW3504.8 : BOOL;
    S367_M_R361_1_로딩완료 AT %MW3501.1 : BOOL;
    S367_M_R366_1_용접가능 AT %MW3504.9 : BOOL;
    S367_M_R366_1_용접완료 AT %MW3501.2 : BOOL;
    S367_M_R369_1_DATA_전송_MEMO AT %MW9015.8 : BOOL; (* S367 M R369 1 DATA 전송 MEMO *)
    S367_M_R369_1_DATA_전송_PLS AT %MW9015.9 : BOOL; (* S367 M R369 1 DATA 전송 PLS *)
    S367_M_R369_1_DATA_전송_SIGN AT %MW9015.10 : BOOL; (* S367 M R369 1 DATA 전송 SIGN *)
    S367_M_R369_1_DATA_전송_완료 AT %MW9015.11 : BOOL; (* S367 M R369 1 DATA 전송 완료 *)
    S367_M_R369_1_언로딩완료 AT %MW3501.3 : BOOL;
    S367_M_RH_AX_CLAMP_전진_LS_이상 AT %MW3610.5 : BOOL; (* S367_M_RH_AX_CLAMP_전진_LS_이상 *)
    S367_M_RH_AX_CLAMP_전진_보조 AT %MW3610.1 : BOOL; (* S367_M_RH_AX_CLAMP_전진_보조 *)
    S367_M_RH_AX_CLAMP_전진단 AT %MW3610.3 : BOOL; (* S367_M_RH_AX_CLAMP_전진단 *)
    S367_M_RH_AX_CLAMP_조건 AT %MW3610.0 : BOOL; (* S367_M_RH_AX_CLAMP_조건 *)
    S367_M_RH_AX_CLAMP_후진_LS_이상 AT %MW3610.6 : BOOL; (* S367_M_RH_AX_CLAMP_후진_LS_이상 *)
    S367_M_RH_AX_CLAMP_후진_보조 AT %MW3610.2 : BOOL; (* S367_M_RH_AX_CLAMP_후진_보조 *)
    S367_M_RH_AX_CLAMP_후진단 AT %MW3610.4 : BOOL; (* S367_M_RH_AX_CLAMP_후진단 *)
    S367_M_RH_AX_LATCH_전진_LS_이상 AT %MW3608.5 : BOOL; (* S367_M_RH_AX_LATCH_전진_LS_이상 *)
    S367_M_RH_AX_LATCH_전진_보조 AT %MW3608.1 : BOOL; (* S367_M_RH_AX_LATCH_전진_보조 *)
    S367_M_RH_AX_LATCH_전진단 AT %MW3608.3 : BOOL; (* S367_M_RH_AX_LATCH_전진단 *)
    S367_M_RH_AX_LATCH_조건 AT %MW3608.0 : BOOL; (* S367_M_RH_AX_LATCH_조건 *)
    S367_M_RH_AX_LATCH_후진_LS_이상 AT %MW3608.6 : BOOL; (* S367_M_RH_AX_LATCH_후진_LS_이상 *)
    S367_M_RH_AX_LATCH_후진_보조 AT %MW3608.2 : BOOL; (* S367_M_RH_AX_LATCH_후진_보조 *)
    S367_M_RH_AX_LATCH_후진단 AT %MW3608.4 : BOOL; (* S367_M_RH_AX_LATCH_후진단 *)
    S367_M_RH_AX_SR_LAT_전진_LS_이상 AT %MW3609.5 : BOOL; (* S367_M_RH_AX_SR_LAT_전진_LS_이상 *)
    S367_M_RH_AX_SR_LAT_전진_보조 AT %MW3609.1 : BOOL; (* S367_M_RH_AX_SR_LAT_전진_보조 *)
    S367_M_RH_AX_SR_LAT_전진단 AT %MW3609.3 : BOOL; (* S367_M_RH_AX_SR_LAT_전진단 *)
    S367_M_RH_AX_SR_LAT_조건 AT %MW3609.0 : BOOL; (* S367_M_RH_AX_SR_LAT_조건 *)
    S367_M_RH_AX_SR_LAT_후진_LS_이상 AT %MW3609.6 : BOOL; (* S367_M_RH_AX_SR_LAT_후진_LS_이상 *)
    S367_M_RH_AX_SR_LAT_후진_보조 AT %MW3609.2 : BOOL; (* S367_M_RH_AX_SR_LAT_후진_보조 *)
    S367_M_RH_AX_SR_LAT_후진단 AT %MW3609.4 : BOOL; (* S367_M_RH_AX_SR_LAT_후진단 *)
    S367_M_RH_CP_OFF AT %MW3517.1 : BOOL; (* S367_M_RH_CP_OFF *)
    S367_M_RH_공기압_이상 AT %MW3513.1 : BOOL; (* S367_M_RH_공기압_이상 *)
    S367_M_S102_간섭무 AT %MW3504.2 : BOOL; (* S367_M_S102_간섭무 *)
    S367_M_SAFETY_불간섭 AT %MW3504.4 : BOOL; (* S367_M_SAFETY_불간섭 *)
    S367_M_SEMI_자동모드 AT %MW3500.2 : BOOL; (* S367_M_SEMI_자동모드 *)
    S367_M_SEQ AT %MW10180 : WORD; (* S367 M SEQ *)
    S367_M_VIN_NO_1_2 AT %MW10191 : WORD; (* S367 M VIN NO 1 2 *)
    S367_M_VIN_NO_3_4 AT %MW10192 : WORD; (* S367 M VIN NO 3 4 *)
    S367_M_VIN_NO_5_6 AT %MW10193 : WORD; (* S367 M VIN NO 5 6 *)
    S367_M_VIN_NO_7_8 AT %MW10194 : WORD; (* S367 M VIN NO 7 8 *)
    S367_M_VIN_NO_9_10 AT %MW10195 : WORD; (* S367 M VIN NO 9 10 *)
    S367_M_공정_FRT_제품감지_무 AT %MW3501.8 : BOOL;
    S367_M_공정_FRT_제품감지_유 AT %MW3501.7 : BOOL;
    S367_M_공정_FRT_제품감지_이상 AT %MW3514.0 : BOOL; (* S367_M_LH_제품감지_이상 *)
    S367_M_공정_RR_제품감지_무 AT %MW3501.10 : BOOL;
    S367_M_공정_RR_제품감지_유 AT %MW3501.9 : BOOL;
    S367_M_공정_RR_제품감지_이상 AT %MW3514.1 : BOOL; (* S367_M_RH_제품감지_이상 *)
    S367_M_공정_SAFETY_NORMAL AT %MW3507.7 : BOOL; (* S367_M_공정_SAFETY_NORMAL *)
    S367_M_공정_불간섭 AT %MW3504.1 : BOOL; (* S367_M_공정_불간섭 *)
    S367_M_공정_원위치 AT %MW3504.0 : BOOL; (* S367_M_공정_원위치 *)
    S367_M_공정_제품감지_무 AT %MW3501.6 : BOOL; (* S367_M_공정_제품감지_무 *)
    S367_M_공정_제품감지_유 AT %MW3501.5 : BOOL; (* S367_M_공정_제품감지_유 *)
    S367_M_공정_차종_무 AT %MW3502.1 : BOOL; (* S367_M_공정_차종_무 *)
    S367_M_공정_차종_보조 AT %MW3502.2 : BOOL; (* S367_M_공정_차종_보조 *)
    S367_M_공정_차종_유 AT %MW3502.0 : BOOL; (* S367_M_공정_차종_유 *)
    S367_M_동작_선택_1 AT %MW3540.0 : BOOL; (* S367_M_동작_선택_1 *)
    S367_M_동작_선택_10 AT %MW3540.9 : BOOL; (* S367_M_동작_선택_10 *)
    S367_M_동작_선택_11 AT %MW3540.10 : BOOL; (* S367_M_동작_선택_11 *)
    S367_M_동작_선택_12 AT %MW3540.11 : BOOL; (* S367_M_동작_선택_12 *)
    S367_M_동작_선택_13 AT %MW3540.12 : BOOL; (* S367_M_동작_선택_13 *)
    S367_M_동작_선택_14 AT %MW3540.13 : BOOL; (* S367_M_동작_선택_14 *)
    S367_M_동작_선택_15 AT %MW3540.14 : BOOL; (* S367_M_동작_선택_15 *)
    S367_M_동작_선택_16 AT %MW3540.15 : BOOL; (* S367_M_동작_선택_16 *)
    S367_M_동작_선택_17 AT %MW3541.0 : BOOL; (* S367_M_동작_선택_17 *)
    S367_M_동작_선택_18 AT %MW3541.1 : BOOL; (* S367_M_동작_선택_18 *)
    S367_M_동작_선택_19 AT %MW3541.2 : BOOL; (* S367_M_동작_선택_19 *)
    S367_M_동작_선택_2 AT %MW3540.1 : BOOL; (* S367_M_동작_선택_2 *)
    S367_M_동작_선택_20 AT %MW3541.3 : BOOL; (* S367_M_동작_선택_20 *)
    S367_M_동작_선택_21 AT %MW3541.4 : BOOL; (* S367_M_동작_선택_21 *)
    S367_M_동작_선택_22 AT %MW3541.5 : BOOL; (* S367_M_동작_선택_22 *)
    S367_M_동작_선택_23 AT %MW3541.6 : BOOL; (* S367_M_동작_선택_23 *)
    S367_M_동작_선택_24 AT %MW3541.7 : BOOL; (* S367_M_동작_선택_24 *)
    S367_M_동작_선택_25 AT %MW3541.8 : BOOL; (* S367_M_동작_선택_25 *)
    S367_M_동작_선택_26 AT %MW3541.9 : BOOL; (* S367_M_동작_선택_26 *)
    S367_M_동작_선택_27 AT %MW3541.10 : BOOL; (* S367_M_동작_선택_27 *)
    S367_M_동작_선택_28 AT %MW3541.11 : BOOL; (* S367_M_동작_선택_28 *)
    S367_M_동작_선택_29 AT %MW3541.12 : BOOL; (* S367_M_동작_선택_29 *)
    S367_M_동작_선택_3 AT %MW3540.2 : BOOL; (* S367_M_동작_선택_3 *)
    S367_M_동작_선택_30 AT %MW3541.13 : BOOL; (* S367_M_동작_선택_30 *)
    S367_M_동작_선택_31 AT %MW3541.14 : BOOL; (* S367_M_동작_선택_31 *)
    S367_M_동작_선택_32 AT %MW3541.15 : BOOL; (* S367_M_동작_선택_32 *)
    S367_M_동작_선택_4 AT %MW3540.3 : BOOL; (* S367_M_동작_선택_4 *)
    S367_M_동작_선택_5 AT %MW3540.4 : BOOL; (* S367_M_동작_선택_5 *)
    S367_M_동작_선택_6 AT %MW3540.5 : BOOL; (* S367_M_동작_선택_6 *)
    S367_M_동작_선택_7 AT %MW3540.6 : BOOL; (* S367_M_동작_선택_7 *)
    S367_M_동작_선택_8 AT %MW3540.7 : BOOL; (* S367_M_동작_선택_8 *)
    S367_M_동작_선택_9 AT %MW3540.8 : BOOL; (* S367_M_동작_선택_9 *)
    S367_M_부저_정지_보조 AT %MW3500.11 : BOOL; (* S367_M_부저_정지_보조 *)
    S367_M_수동모드 AT %MW3500.3 : BOOL; (* S367 선택 수동모드 *)
    S367_M_운전준비_ON AT %MW3500.0 : BOOL; (* S367 운전준비 ON *)
    S367_M_이상_리셋_보조 AT %MW3500.10 : BOOL; (* S367_M_이상_리셋_보조 *)
    S367_M_자동_START AT %MW3500.5 : BOOL; (* S367 자동운전중 *)
    S367_M_자동_운전중 AT %MW3500.4 : BOOL; (* S367 자동운전중 *)
    S367_M_자동모드 AT %MW3500.1 : BOOL; (* S367 선택 자동모드 *)
    S367_M_작업_완료 AT %MW3501.0 : BOOL; (* S367_M_작업_완료 *)
    S367_M_작업완료_SET_PLS AT %MW3500.8 : BOOL; (* S367 M 작업완료 SET PLS *)
    S367_M_작업완료_리셋_PLS AT %MW3500.9 : BOOL; (* S367 M 작업완료 리셋 PLS *)
    S367_M_차종1_AX AT %MW10181.0 : BOOL; (* S367 M 차종1 AX *)
    S367_M_차종1_B AT %MW10181.1 : BOOL; (* S367 M 차종1 B *)
    S367_M_차종1_C AT %MW10181.2 : BOOL; (* S367 M 차종1 C *)
    S367_M_차종1_D AT %MW10181.3 : BOOL; (* S367 M 차종1 D *)
    S367_M_차종1_E AT %MW10181.4 : BOOL; (* S367 M 차종1 E *)
    S367_M_차종1_F AT %MW10181.5 : BOOL; (* S367 M 차종1 F *)
    S367_M_차종1_G AT %MW10181.6 : BOOL; (* S367 M 차종1 G *)
    S367_M_차종1_H AT %MW10181.7 : BOOL; (* S367 M 차종1 H *)
    S367_M_차종2_3DR AT %MW10181.8 : BOOL; (* S367 M 차종2 3DR *)
    S367_M_차종2_4DR AT %MW10181.9 : BOOL; (* S367 M 차종2 4DR *)
    S367_M_차종2_5DR AT %MW10181.10 : BOOL; (* S367 M 차종2 5DR *)
    S367_M_차종2_SP1 AT %MW10181.12 : BOOL; (* S367 M 차종2 SP1 *)
    S367_M_차종2_SP2 AT %MW10181.13 : BOOL; (* S367 M 차종2 SP2 *)
    S367_M_차종2_WGN AT %MW10181.11 : BOOL; (* S367 M 차종2 WGN *)
    S367_M_차종3_LHD AT %MW10181.14 : BOOL; (* S367 M 차종3 LHD *)
    S367_M_차종3_RHD AT %MW10181.15 : BOOL; (* S367 M 차종3 RHD *)
    S367_M_차종4_EEC AT %MW10182.3 : BOOL; (* S367 M 차종4 EEC *)
    S367_M_차종4_SP1 AT %MW10182.8 : BOOL; (* S367 M 차종4 SP1 *)
    S367_M_차종4_SP2 AT %MW10182.9 : BOOL; (* S367 M 차종4 SP2 *)
    S367_M_차종4_SP3 AT %MW10182.11 : BOOL; (* S367 M 차종4 SP3 *)
    S367_M_차종4_SP4 AT %MW10182.12 : BOOL; (* S367 M 차종4 SP4 *)
    S367_M_차종4_SP5 AT %MW10182.13 : BOOL; (* S367 M 차종4 SP5 *)
    S367_M_차종4_SP6 AT %MW10182.14 : BOOL; (* S367 M 차종4 SP6 *)
    S367_M_차종4_SP7 AT %MW10182.15 : BOOL; (* S367 M 차종4 SP7 *)
    S367_M_차종4_내수 AT %MW10182.0 : BOOL; (* S367 M 차종4 내수 *)
    S367_M_차종4_러시아 AT %MW10182.10 : BOOL; (* S367 M 차종4 러시아 *)
    S367_M_차종4_북미 AT %MW10182.2 : BOOL; (* S367 M 차종4 북미 *)
    S367_M_차종4_브라질 AT %MW10182.7 : BOOL; (* S367 M 차종4 브라질 *)
    S367_M_차종4_수출 AT %MW10182.1 : BOOL; (* S367 M 차종4 수출 *)
    S367_M_차종4_중국 AT %MW10182.6 : BOOL; (* S367 M 차종4 중국 *)
    S367_M_차종4_중동 AT %MW10182.5 : BOOL; (* S367 M 차종4 중동 *)
    S367_M_차종4_호주 AT %MW10182.4 : BOOL; (* S367 M 차종4 호주 *)
    S367_M_차종5_AT AT %MW10183.1 : BOOL; (* S367 M 차종5 AT *)
    S367_M_차종5_MT AT %MW10183.0 : BOOL; (* S367 M 차종5 MT *)
    S367_M_차종5_SP1 AT %MW10183.2 : BOOL; (* S367 M 차종5 SP1 *)
    S367_M_차종6_DSROOF AT %MW10183.6 : BOOL; (* S367 M 차종6 DSROOF *)
    S367_M_차종6_SP1 AT %MW10183.7 : BOOL; (* S367 M 차종6 SP1 *)
    S367_M_차종6_썬루프 AT %MW10183.4 : BOOL; (* S367 M 차종6 썬루프 *)
    S367_M_차종6_일반루프 AT %MW10183.3 : BOOL; (* S367 M 차종6 일반루프 *)
    S367_M_차종6_파노라마루프 AT %MW10183.5 : BOOL; (* S367 M 차종6 파노라마루프 *)
    S367_M_차종7_DSL AT %MW10183.9 : BOOL; (* S367 M 차종7 DSL *)
    S367_M_차종7_GSL AT %MW10183.8 : BOOL; (* S367 M 차종7 GSL *)
    S367_M_차종7_SP1 AT %MW10183.10 : BOOL; (* S367 M 차종7 SP1 *)
    S367_M_차종7_SP2 AT %MW10183.11 : BOOL; (* S367 M 차종7 SP2 *)
    S367_M_차종7_SP3 AT %MW10183.12 : BOOL; (* S367 M 차종7 SP3 *)
    S367_M_차종7_SP4 AT %MW10183.13 : BOOL; (* S367 M 차종7 SP4 *)
    S367_M_차종7_SP5 AT %MW10183.14 : BOOL; (* S367 M 차종7 SP5 *)
    S367_M_차종7_SP6 AT %MW10183.15 : BOOL; (* S367 M 차종7 SP6 *)
    S367_M_차종8_2WD AT %MW10184.0 : BOOL; (* S367 M 차종8 2WD *)
    S367_M_차종8_4WD AT %MW10184.1 : BOOL; (* S367 M 차종8 4WD *)
    S367_M_차종8_SP1 AT %MW10184.2 : BOOL; (* S367 M 차종8 SP1 *)
    S367_M_차종9_MPI AT %MW10184.3 : BOOL; (* S367 M 차종9 MPI *)
    S367_M_차종9_SP1 AT %MW10184.5 : BOOL; (* S367 M 차종9 SP1 *)
    S367_M_차종9_SP10 AT %MW10184.14 : BOOL; (* S367 M 차종9 SP10 *)
    S367_M_차종9_SP11 AT %MW10184.15 : BOOL; (* S367 M 차종9 SP11 *)
    S367_M_차종9_SP2 AT %MW10184.6 : BOOL; (* S367 M 차종9 SP2 *)
    S367_M_차종9_SP3 AT %MW10184.7 : BOOL; (* S367 M 차종9 SP3 *)
    S367_M_차종9_SP4 AT %MW10184.8 : BOOL; (* S367 M 차종9 SP4 *)
    S367_M_차종9_SP5 AT %MW10184.9 : BOOL; (* S367 M 차종9 SP5 *)
    S367_M_차종9_SP6 AT %MW10184.10 : BOOL; (* S367 M 차종9 SP6 *)
    S367_M_차종9_SP7 AT %MW10184.11 : BOOL; (* S367 M 차종9 SP7 *)
    S367_M_차종9_SP8 AT %MW10184.12 : BOOL; (* S367 M 차종9 SP8 *)
    S367_M_차종9_SP9 AT %MW10184.13 : BOOL; (* S367 M 차종9 SP9 *)
    S367_M_차종9_T_GDI AT %MW10184.4 : BOOL; (* S367 M 차종9 T GDI *)
    S367_M_차종_AS AT %MW10190.9 : BOOL; (* S367 M 차종 AS *)
    S367_M_차종_OPT1_R_RACK_무 AT %MW10185.3 : BOOL; (* S367 M 차종 OPT1 R RACK 무 *)
    S367_M_차종_OPT1_R_RACK_유 AT %MW10185.2 : BOOL; (* S367 M 차종 OPT1 R RACK 유 *)
    S367_M_차종_OPT1_SP1 AT %MW10185.10 : BOOL; (* S367 M 차종 OPT1 SP1 *)
    S367_M_차종_OPT1_SP2 AT %MW10185.11 : BOOL; (* S367 M 차종 OPT1 SP2 *)
    S367_M_차종_OPT1_SP3 AT %MW10185.12 : BOOL; (* S367 M 차종 OPT1 SP3 *)
    S367_M_차종_OPT1_SP4 AT %MW10185.13 : BOOL; (* S367 M 차종 OPT1 SP4 *)
    S367_M_차종_OPT1_SP5 AT %MW10185.14 : BOOL; (* S367 M 차종 OPT1 SP5 *)
    S367_M_차종_OPT1_SP6 AT %MW10185.15 : BOOL; (* S367 M 차종 OPT1 SP6 *)
    S367_M_차종_OPT1_S_REP_EATER_무 AT %MW10185.7 : BOOL; (* S367 M 차종 OPT1 S REP EATER 무 *)
    S367_M_차종_OPT1_S_REP_EATER_유 AT %MW10185.6 : BOOL; (* S367 M 차종 OPT1 S REP EATER 유 *)
    S367_M_차종_OPT1_VAN_무 AT %MW10185.9 : BOOL; (* S367 M 차종 OPT1 VAN 무 *)
    S367_M_차종_OPT1_VAN_유 AT %MW10185.8 : BOOL; (* S367 M 차종 OPT1 VAN 유 *)
    S367_M_차종_OPT1_슬라이딩_무 AT %MW10185.1 : BOOL; (* S367 M 차종 OPT1 슬라이딩 무 *)
    S367_M_차종_OPT1_슬라이딩_유 AT %MW10185.0 : BOOL; (* S367 M 차종 OPT1 슬라이딩 유 *)
    S367_M_차종_OPT1_폴딩_무 AT %MW10185.5 : BOOL; (* S367 M 차종 OPT1 폴딩 무 *)
    S367_M_차종_OPT1_폴딩_유 AT %MW10185.4 : BOOL; (* S367 M 차종 OPT1 폴딩 유 *)
    S367_M_차종_OPT2_SP_WORD1 AT %MW10186 : WORD; (* S367 M 차종 OPT2 SP WORD1 *)
    S367_M_차종_OPT3_SP_WORD2 AT %MW10187 : WORD; (* S367 M 차종 OPT3 SP WORD2 *)
    S367_M_차종_OPT4_SP_WORD3 AT %MW10188 : WORD; (* S367 M 차종 OPT4 SP WORD3 *)
    S367_M_차종_OPT5_SP_WORD4 AT %MW10189 : WORD; (* S367 M 차종 OPT5 SP WORD4 *)
    S367_M_차종_SP1 AT %MW10190.0 : BOOL; (* S367 M 차종 SP1 *)
    S367_M_차종_SP2 AT %MW10190.1 : BOOL; (* S367 M 차종 SP2 *)
    S367_M_차종_SP3 AT %MW10190.2 : BOOL; (* S367 M 차종 SP3 *)
    S367_M_차종_SP4 AT %MW10190.3 : BOOL; (* S367 M 차종 SP4 *)
    S367_M_차종_SP5 AT %MW10190.4 : BOOL; (* S367 M 차종 SP5 *)
    S367_M_차종_SP6 AT %MW10190.5 : BOOL; (* S367 M 차종 SP6 *)
    S367_M_차종_SP7 AT %MW10190.6 : BOOL; (* S367 M 차종 SP7 *)
    S367_M_차종_SP8 AT %MW10190.7 : BOOL; (* S367 M 차종 SP8 *)
    S367_M_차종_SP9 AT %MW10190.15 : BOOL; (* S367 M 차종 SP9 *)
    S367_M_차종_공대차 AT %MW10190.12 : BOOL; (* S367 M 차종 공대차 *)
    S367_M_차종_공차 AT %MW10190.10 : BOOL; (* S367 M 차종 공차 *)
    S367_M_차종_불량대차 AT %MW10190.13 : BOOL; (* S367 M 차종 불량대차 *)
    S367_M_차종_불량차 AT %MW10190.11 : BOOL; (* S367 M 차종 불량차 *)
    S367_M_차종_비축 AT %MW10190.8 : BOOL; (* S367 M 차종 비축 *)
    S367_M_차종_취출대차 AT %MW10190.14 : BOOL; (* S367 M 차종 취출대차 *)
    S367_M_총괄_CP_이상 AT %MW3509.7 : BOOL; (* S367 CP OFF 이상 *)
    S367_M_총괄_CT_이상 AT %MW3510.4 : BOOL; (* S367   TACK TIME 이상 *)
    S367_M_총괄_EOCR_이상 AT %MW3509.8 : BOOL; (* S367_M_총괄_EOCR_이상 *)
    S367_M_총괄_INV_이상 AT %MW3509.9 : BOOL; (* S367_M_총괄_INV_이상 *)
    S367_M_총괄_LS_이상 AT %MW3509.15 : BOOL; (* S367 LS 이상 *)
    S367_M_총괄_MATCH_이상 AT %MW3510.0 : BOOL; (* S367 매트SW 이상 *)
    S367_M_총괄_MC_이상 AT %MW3509.13 : BOOL; (* S367_M_총괄_MC_이상 *)
    S367_M_총괄_MOTOR_이상 AT %MW3510.3 : BOOL; (* S367_M_총괄_MOTOR_이상 *)
    S367_M_총괄_NFB_이상 AT %MW3509.11 : BOOL; (* S367_M_총괄_NFB_이상 *)
    S367_M_총괄_ROBOT_이상 AT %MW3510.1 : BOOL; (* S367 ROBOT 이상 *)
    S367_M_총괄_SAFETY_이상 AT %MW3509.2 : BOOL; (* S367_M_총괄_SAFETY_이상 *)
    S367_M_총괄_SRV_이상 AT %MW3509.10 : BOOL; (* S367_M_총괄_SRV_이상 *)
    S367_M_총괄_공기압_이상 AT %MW3509.3 : BOOL; (* S367 공기압 이상 *)
    S367_M_총괄_비상정지_이상 AT %MW3509.1 : BOOL; (* S367_M_총괄_비상정지_이상 *)
    S367_M_총괄_사양_이상 AT %MW3509.6 : BOOL; (* S367 사양 이상 *)
    S367_M_총괄_오버런_이상 AT %MW3509.12 : BOOL; (* S367_M_총괄_오버런_이상 *)
    S367_M_총괄_용접타점수_이상 AT %MW3510.2 : BOOL; (* S367 용접타점수 이상 *)
    S367_M_총괄_이상 AT %MW3509.0 : BOOL; (* S367_M_총괄_이상 *)
    S367_M_총괄_제품감지_이상 AT %MW3509.4 : BOOL; (* S367 제품감지 이상 *)
    S367_M_총괄_차종_이상 AT %MW3509.5 : BOOL; (* S367 차종 이상 *)
    S367_M_총괄_통신_이상 AT %MW3509.14 : BOOL; (* S367 통신이상 *)
    S367_RH_M_NODE_6_20_통신_이상 AT %MW3524.1 : BOOL;
    S367_전진_ON AT %MW3548.1 : BOOL; (* S367_전진_ON *)
    S367_후진_ON AT %MW3548.2 : BOOL; (* S367_후진_ON *)
    S368_HOME AT %MW4048.0 : BOOL; (* S368_HOME *)
    S368_LH_M_NODE_6_31_통신_이상 AT %MW4024.0 : BOOL;
    S368_M_BYPASS_보조 AT %MW4003.15 : BOOL; (* S368 M BYPASS 보조 *)
    S368_M_CTIME_OVER_ALRAM AT %MW4007.14 : BOOL; (* S368_M_CTIME_OVER_ALRAM *)
    S368_M_CTIME_OVER_MUTE AT %MW4007.13 : BOOL; (* S368_M_CTIME_OVER_MUTE *)
    S368_M_DATA_삭제_PLS AT %MW9016.0 : BOOL; (* S368 M DATA 삭제 PLS *)
    S368_M_DATA_삭제_SIGN AT %MW9016.1 : BOOL; (* S368 M DATA 삭제 SIGN *)
    S368_M_DATA_삭제_완료 AT %MW9016.2 : BOOL; (* S368 M DATA 삭제 완료 *)
    S368_M_HANGER_CLP_전진_LS_이상 AT %MW4111.5 : BOOL; (* S368_M_HANGER_CLP_전진_LS_이상 *)
    S368_M_HANGER_CLP_전진_보조 AT %MW4111.1 : BOOL; (* S368_M_HANGER_CLP_전진_보조 *)
    S368_M_HANGER_CLP_전진단 AT %MW4111.3 : BOOL; (* S368_M_HANGER_CLP_전진단 *)
    S368_M_HANGER_CLP_조건 AT %MW4111.0 : BOOL; (* S368_M_HANGER_CLP_조건 *)
    S368_M_HANGER_CLP_후진_LS_이상 AT %MW4111.6 : BOOL; (* S368_M_HANGER_CLP_후진_LS_이상 *)
    S368_M_HANGER_CLP_후진_보조 AT %MW4111.2 : BOOL; (* S368_M_HANGER_CLP_후진_보조 *)
    S368_M_HANGER_CLP_후진단 AT %MW4111.4 : BOOL; (* S368_M_HANGER_CLP_후진단 *)
    S368_M_HANGER_급전급기_ADV_AUX AT %MW4103.1 : BOOL;
    S368_M_HANGER_급전급기_COND AT %MW4103.0 : BOOL;
    S368_M_HANGER_급전급기_RET_AUX AT %MW4103.2 : BOOL;
    S368_M_HANGER_급전급기_전진_LS_이상 AT %MW4103.5 : BOOL;
    S368_M_HANGER_급전급기_전진단 AT %MW4103.3 : BOOL;
    S368_M_HANGER_급전급기_후진_LS_이상 AT %MW4103.6 : BOOL;
    S368_M_HANGER_급전급기_후진단 AT %MW4103.4 : BOOL;
    S368_M_LC_정상 AT %MW4007.5 : BOOL; (* S368_M_LC_정상 *)
    S368_M_LH_AX_CLAMP_전진_LS_이상 AT %MW4102.5 : BOOL; (* S368_M_LH_AX_CLAMP_전진_LS_이상 *)
    S368_M_LH_AX_CLAMP_전진_보조 AT %MW4102.1 : BOOL; (* S368_M_LH_AX_CLAMP_전진_보조 *)
    S368_M_LH_AX_CLAMP_전진단 AT %MW4102.3 : BOOL; (* S368_M_LH_AX_CLAMP_전진단 *)
    S368_M_LH_AX_CLAMP_조건 AT %MW4102.0 : BOOL; (* S368_M_LH_AX_CLAMP_조건 *)
    S368_M_LH_AX_CLAMP_후진_LS_이상 AT %MW4102.6 : BOOL; (* S368_M_LH_AX_CLAMP_후진_LS_이상 *)
    S368_M_LH_AX_CLAMP_후진_보조 AT %MW4102.2 : BOOL; (* S368_M_LH_AX_CLAMP_후진_보조 *)
    S368_M_LH_AX_CLAMP_후진단 AT %MW4102.4 : BOOL; (* S368_M_LH_AX_CLAMP_후진단 *)
    S368_M_LH_AX_LATCH_전진_LS_이상 AT %MW4100.5 : BOOL; (* S368_M_LH_AX_LATCH_전진_LS_이상 *)
    S368_M_LH_AX_LATCH_전진_보조 AT %MW4100.1 : BOOL; (* S368_M_LH_AX_LATCH_전진_보조 *)
    S368_M_LH_AX_LATCH_전진단 AT %MW4100.3 : BOOL; (* S368_M_LH_AX_LATCH_전진단 *)
    S368_M_LH_AX_LATCH_조건 AT %MW4100.0 : BOOL; (* S368_M_LH_AX_LATCH_조건 *)
    S368_M_LH_AX_LATCH_후진_LS_이상 AT %MW4100.6 : BOOL; (* S368_M_LH_AX_LATCH_후진_LS_이상 *)
    S368_M_LH_AX_LATCH_후진_보조 AT %MW4100.2 : BOOL; (* S368_M_LH_AX_LATCH_후진_보조 *)
    S368_M_LH_AX_LATCH_후진단 AT %MW4100.4 : BOOL; (* S368_M_LH_AX_LATCH_후진단 *)
    S368_M_LH_AX_SR_LAT_전진_LS_이상 AT %MW4101.5 : BOOL; (* S368_M_LH_AX_SR_LAT_전진_LS_이상 *)
    S368_M_LH_AX_SR_LAT_전진_보조 AT %MW4101.1 : BOOL; (* S368_M_LH_AX_SR_LAT_전진_보조 *)
    S368_M_LH_AX_SR_LAT_전진단 AT %MW4101.3 : BOOL; (* S368_M_LH_AX_SR_LAT_전진단 *)
    S368_M_LH_AX_SR_LAT_조건 AT %MW4101.0 : BOOL; (* S368_M_LH_AX_SR_LAT_조건 *)
    S368_M_LH_AX_SR_LAT_후진_LS_이상 AT %MW4101.6 : BOOL; (* S368_M_LH_AX_SR_LAT_후진_LS_이상 *)
    S368_M_LH_AX_SR_LAT_후진_보조 AT %MW4101.2 : BOOL; (* S368_M_LH_AX_SR_LAT_후진_보조 *)
    S368_M_LH_AX_SR_LAT_후진단 AT %MW4101.4 : BOOL; (* S368_M_LH_AX_SR_LAT_후진단 *)
    S368_M_LH_CP_OFF AT %MW4017.0 : BOOL; (* S368_M_LH_CP_OFF *)
    S368_M_LH_공기압_이상 AT %MW4013.0 : BOOL; (* S368_M_LH_공기압_이상 *)
    S368_M_MAT_정상 AT %MW4007.6 : BOOL; (* S368_M_MAT_정상 *)
    S368_M_OP_ESTOP_NORMAL AT %MW4007.1 : BOOL; (* S368_M_OP_ESTOP_NORMAL *)
    S368_M_R368_1_해밍가능 AT %MW4004.10 : BOOL;
    S368_M_R368_1_행거안착가능 AT %MW4004.9 : BOOL;
    S368_M_R368_1_행거안착완료 AT %MW4001.2 : BOOL;
    S368_M_R368_1_헤밍완료 AT %MW4001.3 : BOOL;
    S368_M_R369_1_안착가능 AT %MW4004.8 : BOOL;
    S368_M_R369_1_안착완료 AT %MW4001.1 : BOOL;
    S368_M_R369_1_언로딩완료 AT %MW4001.4 : BOOL;
    S368_M_RH_AX_CLAMP_전진_LS_이상 AT %MW4110.5 : BOOL; (* S368_M_RH_AX_CLAMP_전진_LS_이상 *)
    S368_M_RH_AX_CLAMP_전진_보조 AT %MW4110.1 : BOOL; (* S368_M_RH_AX_CLAMP_전진_보조 *)
    S368_M_RH_AX_CLAMP_전진단 AT %MW4110.3 : BOOL; (* S368_M_RH_AX_CLAMP_전진단 *)
    S368_M_RH_AX_CLAMP_조건 AT %MW4110.0 : BOOL; (* S368_M_RH_AX_CLAMP_조건 *)
    S368_M_RH_AX_CLAMP_후진_LS_이상 AT %MW4110.6 : BOOL; (* S368_M_RH_AX_CLAMP_후진_LS_이상 *)
    S368_M_RH_AX_CLAMP_후진_보조 AT %MW4110.2 : BOOL; (* S368_M_RH_AX_CLAMP_후진_보조 *)
    S368_M_RH_AX_CLAMP_후진단 AT %MW4110.4 : BOOL; (* S368_M_RH_AX_CLAMP_후진단 *)
    S368_M_RH_AX_LATCH_전진_LS_이상 AT %MW4108.5 : BOOL; (* S368_M_RH_AX_LATCH_전진_LS_이상 *)
    S368_M_RH_AX_LATCH_전진_보조 AT %MW4108.1 : BOOL; (* S368_M_RH_AX_LATCH_전진_보조 *)
    S368_M_RH_AX_LATCH_전진단 AT %MW4108.3 : BOOL; (* S368_M_RH_AX_LATCH_전진단 *)
    S368_M_RH_AX_LATCH_조건 AT %MW4108.0 : BOOL; (* S368_M_RH_AX_LATCH_조건 *)
    S368_M_RH_AX_LATCH_후진_LS_이상 AT %MW4108.6 : BOOL; (* S368_M_RH_AX_LATCH_후진_LS_이상 *)
    S368_M_RH_AX_LATCH_후진_보조 AT %MW4108.2 : BOOL; (* S368_M_RH_AX_LATCH_후진_보조 *)
    S368_M_RH_AX_LATCH_후진단 AT %MW4108.4 : BOOL; (* S368_M_RH_AX_LATCH_후진단 *)
    S368_M_RH_AX_SR_LAT_전진_LS_이상 AT %MW4109.5 : BOOL; (* S368_M_RH_AX_SR_LAT_전진_LS_이상 *)
    S368_M_RH_AX_SR_LAT_전진_보조 AT %MW4109.1 : BOOL; (* S368_M_RH_AX_SR_LAT_전진_보조 *)
    S368_M_RH_AX_SR_LAT_전진단 AT %MW4109.3 : BOOL; (* S368_M_RH_AX_SR_LAT_전진단 *)
    S368_M_RH_AX_SR_LAT_조건 AT %MW4109.0 : BOOL; (* S368_M_RH_AX_SR_LAT_조건 *)
    S368_M_RH_AX_SR_LAT_후진_LS_이상 AT %MW4109.6 : BOOL; (* S368_M_RH_AX_SR_LAT_후진_LS_이상 *)
    S368_M_RH_AX_SR_LAT_후진_보조 AT %MW4109.2 : BOOL; (* S368_M_RH_AX_SR_LAT_후진_보조 *)
    S368_M_RH_AX_SR_LAT_후진단 AT %MW4109.4 : BOOL; (* S368_M_RH_AX_SR_LAT_후진단 *)
    S368_M_RH_CP_OFF AT %MW4017.1 : BOOL; (* S368_M_RH_CP_OFF *)
    S368_M_RH_공기압_이상 AT %MW4013.1 : BOOL; (* S368_M_RH_공기압_이상 *)
    S368_M_S102_간섭무 AT %MW4004.2 : BOOL; (* S368_M_S102_간섭무 *)
    S368_M_S369_1_DATA_전송_MEMO AT %MW9016.8 : BOOL; (* S368 M S369 1 DATA 전송 MEMO *)
    S368_M_S369_1_DATA_전송_PLS AT %MW9016.9 : BOOL; (* S368 M S369 1 DATA 전송 PLS *)
    S368_M_S369_1_DATA_전송_SIGN AT %MW9016.10 : BOOL; (* S368 M S369 1 DATA 전송 SIGN *)
    S368_M_S369_1_DATA_전송_완료 AT %MW9016.11 : BOOL; (* S368 M S369 1 DATA 전송 완료 *)
    S368_M_SAFETY_불간섭 AT %MW4004.4 : BOOL; (* S368_M_SAFETY_불간섭 *)
    S368_M_SEMI_자동모드 AT %MW4000.2 : BOOL; (* S368_M_SEMI_자동모드 *)
    S368_M_SEQ AT %MW10200 : WORD; (* S368 M SEQ *)
    S368_M_VIN_NO_1_2 AT %MW10211 : WORD; (* S368 M VIN NO 1 2 *)
    S368_M_VIN_NO_3_4 AT %MW10212 : WORD; (* S368 M VIN NO 3 4 *)
    S368_M_VIN_NO_5_6 AT %MW10213 : WORD; (* S368 M VIN NO 5 6 *)
    S368_M_VIN_NO_7_8 AT %MW10214 : WORD; (* S368 M VIN NO 7 8 *)
    S368_M_VIN_NO_9_10 AT %MW10215 : WORD; (* S368 M VIN NO 9 10 *)
    S368_M_공정_FRT_제품감지_무 AT %MW4001.8 : BOOL;
    S368_M_공정_FRT_제품감지_유 AT %MW4001.7 : BOOL;
    S368_M_공정_FRT_제품감지_이상 AT %MW4014.0 : BOOL;
    S368_M_공정_HANGER_감지_무 AT %MW4001.12 : BOOL;
    S368_M_공정_HANGER_감지_유 AT %MW4001.11 : BOOL;
    S368_M_공정_HANGER_감지_이상 AT %MW4014.2 : BOOL;
    S368_M_공정_RR_제품감지_무 AT %MW4001.10 : BOOL;
    S368_M_공정_RR_제품감지_유 AT %MW4001.9 : BOOL;
    S368_M_공정_RR_제품감지_이상 AT %MW4014.1 : BOOL;
    S368_M_공정_SAFETY_NORMAL AT %MW4007.7 : BOOL; (* S368_M_공정_SAFETY_NORMAL *)
    S368_M_공정_불간섭 AT %MW4004.1 : BOOL; (* S368_M_공정_불간섭 *)
    S368_M_공정_원위치 AT %MW4004.0 : BOOL; (* S368_M_공정_원위치 *)
    S368_M_공정_제품감지_무 AT %MW4001.6 : BOOL; (* S368_M_공정_제품감지_무 *)
    S368_M_공정_제품감지_유 AT %MW4001.5 : BOOL; (* S368_M_공정_제품감지_유 *)
    S368_M_공정_차종_무 AT %MW4002.1 : BOOL; (* S368_M_공정_차종_무 *)
    S368_M_공정_차종_유 AT %MW4002.0 : BOOL; (* S368_M_공정_차종_유 *)
    S368_M_동작_선택_1 AT %MW4040.0 : BOOL; (* S368_M_동작_선택_1 *)
    S368_M_동작_선택_10 AT %MW4040.9 : BOOL; (* S368_M_동작_선택_10 *)
    S368_M_동작_선택_11 AT %MW4040.10 : BOOL; (* S368_M_동작_선택_11 *)
    S368_M_동작_선택_12 AT %MW4040.11 : BOOL; (* S368_M_동작_선택_12 *)
    S368_M_동작_선택_13 AT %MW4040.12 : BOOL; (* S368_M_동작_선택_13 *)
    S368_M_동작_선택_14 AT %MW4040.13 : BOOL; (* S368_M_동작_선택_14 *)
    S368_M_동작_선택_15 AT %MW4040.14 : BOOL; (* S368_M_동작_선택_15 *)
    S368_M_동작_선택_16 AT %MW4040.15 : BOOL; (* S368_M_동작_선택_16 *)
    S368_M_동작_선택_17 AT %MW4041.0 : BOOL; (* S368_M_동작_선택_17 *)
    S368_M_동작_선택_18 AT %MW4041.1 : BOOL; (* S368_M_동작_선택_18 *)
    S368_M_동작_선택_19 AT %MW4041.2 : BOOL; (* S368_M_동작_선택_19 *)
    S368_M_동작_선택_2 AT %MW4040.1 : BOOL; (* S368_M_동작_선택_2 *)
    S368_M_동작_선택_20 AT %MW4041.3 : BOOL; (* S368_M_동작_선택_20 *)
    S368_M_동작_선택_21 AT %MW4041.4 : BOOL; (* S368_M_동작_선택_21 *)
    S368_M_동작_선택_22 AT %MW4041.5 : BOOL; (* S368_M_동작_선택_22 *)
    S368_M_동작_선택_23 AT %MW4041.6 : BOOL; (* S368_M_동작_선택_23 *)
    S368_M_동작_선택_24 AT %MW4041.7 : BOOL; (* S368_M_동작_선택_24 *)
    S368_M_동작_선택_25 AT %MW4041.8 : BOOL; (* S368_M_동작_선택_25 *)
    S368_M_동작_선택_26 AT %MW4041.9 : BOOL; (* S368_M_동작_선택_26 *)
    S368_M_동작_선택_27 AT %MW4041.10 : BOOL; (* S368_M_동작_선택_27 *)
    S368_M_동작_선택_28 AT %MW4041.11 : BOOL; (* S368_M_동작_선택_28 *)
    S368_M_동작_선택_29 AT %MW4041.12 : BOOL; (* S368_M_동작_선택_29 *)
    S368_M_동작_선택_3 AT %MW4040.2 : BOOL; (* S368_M_동작_선택_3 *)
    S368_M_동작_선택_30 AT %MW4041.13 : BOOL; (* S368_M_동작_선택_30 *)
    S368_M_동작_선택_31 AT %MW4041.14 : BOOL; (* S368_M_동작_선택_31 *)
    S368_M_동작_선택_32 AT %MW4041.15 : BOOL; (* S368_M_동작_선택_32 *)
    S368_M_동작_선택_4 AT %MW4040.3 : BOOL; (* S368_M_동작_선택_4 *)
    S368_M_동작_선택_5 AT %MW4040.4 : BOOL; (* S368_M_동작_선택_5 *)
    S368_M_동작_선택_6 AT %MW4040.5 : BOOL; (* S368_M_동작_선택_6 *)
    S368_M_동작_선택_7 AT %MW4040.6 : BOOL; (* S368_M_동작_선택_7 *)
    S368_M_동작_선택_8 AT %MW4040.7 : BOOL; (* S368_M_동작_선택_8 *)
    S368_M_동작_선택_9 AT %MW4040.8 : BOOL; (* S368_M_동작_선택_9 *)
    S368_M_부저_정지_보조 AT %MW4000.11 : BOOL; (* S368_M_부저_정지_보조 *)
    S368_M_수동모드 AT %MW4000.3 : BOOL; (* S368 선택 수동모드 *)
    S368_M_운전준비_ON AT %MW4000.0 : BOOL; (* S368 운전준비 ON *)
    S368_M_이상_리셋_보조 AT %MW4000.10 : BOOL; (* S368_M_이상_리셋_보조 *)
    S368_M_자동_START AT %MW4000.5 : BOOL; (* S368 자동운전중 *)
    S368_M_자동_운전중 AT %MW4000.4 : BOOL; (* S368 자동운전중 *)
    S368_M_자동모드 AT %MW4000.1 : BOOL; (* S368 선택 자동모드 *)
    S368_M_작업_완료 AT %MW4001.0 : BOOL; (* S368_M_작업_완료 *)
    S368_M_작업완료_SET_PLS AT %MW4000.8 : BOOL; (* S368 M 작업완료 SET PLS *)
    S368_M_작업완료_리셋_PLS AT %MW4000.9 : BOOL; (* S368 M 작업완료 리셋 PLS *)
    S368_M_차종1_AX AT %MW10201.0 : BOOL; (* S368 M 차종1 AX *)
    S368_M_차종1_B AT %MW10201.1 : BOOL; (* S368 M 차종1 B *)
    S368_M_차종1_C AT %MW10201.2 : BOOL; (* S368 M 차종1 C *)
    S368_M_차종1_D AT %MW10201.3 : BOOL; (* S368 M 차종1 D *)
    S368_M_차종1_E AT %MW10201.4 : BOOL; (* S368 M 차종1 E *)
    S368_M_차종1_F AT %MW10201.5 : BOOL; (* S368 M 차종1 F *)
    S368_M_차종1_G AT %MW10201.6 : BOOL; (* S368 M 차종1 G *)
    S368_M_차종1_H AT %MW10201.7 : BOOL; (* S368 M 차종1 H *)
    S368_M_차종2_3DR AT %MW10201.8 : BOOL; (* S368 M 차종2 3DR *)
    S368_M_차종2_4DR AT %MW10201.9 : BOOL; (* S368 M 차종2 4DR *)
    S368_M_차종2_5DR AT %MW10201.10 : BOOL; (* S368 M 차종2 5DR *)
    S368_M_차종2_SP1 AT %MW10201.12 : BOOL; (* S368 M 차종2 SP1 *)
    S368_M_차종2_SP2 AT %MW10201.13 : BOOL; (* S368 M 차종2 SP2 *)
    S368_M_차종2_WGN AT %MW10201.11 : BOOL; (* S368 M 차종2 WGN *)
    S368_M_차종3_LHD AT %MW10201.14 : BOOL; (* S368 M 차종3 LHD *)
    S368_M_차종3_RHD AT %MW10201.15 : BOOL; (* S368 M 차종3 RHD *)
    S368_M_차종4_EEC AT %MW10202.3 : BOOL; (* S368 M 차종4 EEC *)
    S368_M_차종4_SP1 AT %MW10202.8 : BOOL; (* S368 M 차종4 SP1 *)
    S368_M_차종4_SP2 AT %MW10202.9 : BOOL; (* S368 M 차종4 SP2 *)
    S368_M_차종4_SP3 AT %MW10202.11 : BOOL; (* S368 M 차종4 SP3 *)
    S368_M_차종4_SP4 AT %MW10202.12 : BOOL; (* S368 M 차종4 SP4 *)
    S368_M_차종4_SP5 AT %MW10202.13 : BOOL; (* S368 M 차종4 SP5 *)
    S368_M_차종4_SP6 AT %MW10202.14 : BOOL; (* S368 M 차종4 SP6 *)
    S368_M_차종4_SP7 AT %MW10202.15 : BOOL; (* S368 M 차종4 SP7 *)
    S368_M_차종4_내수 AT %MW10202.0 : BOOL; (* S368 M 차종4 내수 *)
    S368_M_차종4_러시아 AT %MW10202.10 : BOOL; (* S368 M 차종4 러시아 *)
    S368_M_차종4_북미 AT %MW10202.2 : BOOL; (* S368 M 차종4 북미 *)
    S368_M_차종4_브라질 AT %MW10202.7 : BOOL; (* S368 M 차종4 브라질 *)
    S368_M_차종4_수출 AT %MW10202.1 : BOOL; (* S368 M 차종4 수출 *)
    S368_M_차종4_중국 AT %MW10202.6 : BOOL; (* S368 M 차종4 중국 *)
    S368_M_차종4_중동 AT %MW10202.5 : BOOL; (* S368 M 차종4 중동 *)
    S368_M_차종4_호주 AT %MW10202.4 : BOOL; (* S368 M 차종4 호주 *)
    S368_M_차종5_AT AT %MW10203.1 : BOOL; (* S368 M 차종5 AT *)
    S368_M_차종5_MT AT %MW10203.0 : BOOL; (* S368 M 차종5 MT *)
    S368_M_차종5_SP1 AT %MW10203.2 : BOOL; (* S368 M 차종5 SP1 *)
    S368_M_차종6_DSROOF AT %MW10203.6 : BOOL; (* S368 M 차종6 DSROOF *)
    S368_M_차종6_SP1 AT %MW10203.7 : BOOL; (* S368 M 차종6 SP1 *)
    S368_M_차종6_썬루프 AT %MW10203.4 : BOOL; (* S368 M 차종6 썬루프 *)
    S368_M_차종6_일반루프 AT %MW10203.3 : BOOL; (* S368 M 차종6 일반루프 *)
    S368_M_차종6_파노라마루프 AT %MW10203.5 : BOOL; (* S368 M 차종6 파노라마루프 *)
    S368_M_차종7_DSL AT %MW10203.9 : BOOL; (* S368 M 차종7 DSL *)
    S368_M_차종7_GSL AT %MW10203.8 : BOOL; (* S368 M 차종7 GSL *)
    S368_M_차종7_SP1 AT %MW10203.10 : BOOL; (* S368 M 차종7 SP1 *)
    S368_M_차종7_SP2 AT %MW10203.11 : BOOL; (* S368 M 차종7 SP2 *)
    S368_M_차종7_SP3 AT %MW10203.12 : BOOL; (* S368 M 차종7 SP3 *)
    S368_M_차종7_SP4 AT %MW10203.13 : BOOL; (* S368 M 차종7 SP4 *)
    S368_M_차종7_SP5 AT %MW10203.14 : BOOL; (* S368 M 차종7 SP5 *)
    S368_M_차종7_SP6 AT %MW10203.15 : BOOL; (* S368 M 차종7 SP6 *)
    S368_M_차종8_2WD AT %MW10204.0 : BOOL; (* S368 M 차종8 2WD *)
    S368_M_차종8_4WD AT %MW10204.1 : BOOL; (* S368 M 차종8 4WD *)
    S368_M_차종8_SP1 AT %MW10204.2 : BOOL; (* S368 M 차종8 SP1 *)
    S368_M_차종9_MPI AT %MW10204.3 : BOOL; (* S368 M 차종9 MPI *)
    S368_M_차종9_SP1 AT %MW10204.5 : BOOL; (* S368 M 차종9 SP1 *)
    S368_M_차종9_SP10 AT %MW10204.14 : BOOL; (* S368 M 차종9 SP10 *)
    S368_M_차종9_SP11 AT %MW10204.15 : BOOL; (* S368 M 차종9 SP11 *)
    S368_M_차종9_SP2 AT %MW10204.6 : BOOL; (* S368 M 차종9 SP2 *)
    S368_M_차종9_SP3 AT %MW10204.7 : BOOL; (* S368 M 차종9 SP3 *)
    S368_M_차종9_SP4 AT %MW10204.8 : BOOL; (* S368 M 차종9 SP4 *)
    S368_M_차종9_SP5 AT %MW10204.9 : BOOL; (* S368 M 차종9 SP5 *)
    S368_M_차종9_SP6 AT %MW10204.10 : BOOL; (* S368 M 차종9 SP6 *)
    S368_M_차종9_SP7 AT %MW10204.11 : BOOL; (* S368 M 차종9 SP7 *)
    S368_M_차종9_SP8 AT %MW10204.12 : BOOL; (* S368 M 차종9 SP8 *)
    S368_M_차종9_SP9 AT %MW10204.13 : BOOL; (* S368 M 차종9 SP9 *)
    S368_M_차종9_T_GDI AT %MW10204.4 : BOOL; (* S368 M 차종9 T GDI *)
    S368_M_차종_AS AT %MW10210.9 : BOOL; (* S368 M 차종 AS *)
    S368_M_차종_OPT1_R_RACK_무 AT %MW10205.3 : BOOL; (* S368 M 차종 OPT1 R RACK 무 *)
    S368_M_차종_OPT1_R_RACK_유 AT %MW10205.2 : BOOL; (* S368 M 차종 OPT1 R RACK 유 *)
    S368_M_차종_OPT1_SP1 AT %MW10205.10 : BOOL; (* S368 M 차종 OPT1 SP1 *)
    S368_M_차종_OPT1_SP2 AT %MW10205.11 : BOOL; (* S368 M 차종 OPT1 SP2 *)
    S368_M_차종_OPT1_SP3 AT %MW10205.12 : BOOL; (* S368 M 차종 OPT1 SP3 *)
    S368_M_차종_OPT1_SP4 AT %MW10205.13 : BOOL; (* S368 M 차종 OPT1 SP4 *)
    S368_M_차종_OPT1_SP5 AT %MW10205.14 : BOOL; (* S368 M 차종 OPT1 SP5 *)
    S368_M_차종_OPT1_SP6 AT %MW10205.15 : BOOL; (* S368 M 차종 OPT1 SP6 *)
    S368_M_차종_OPT1_S_REP_EATER_무 AT %MW10205.7 : BOOL; (* S368 M 차종 OPT1 S REP EATER 무 *)
    S368_M_차종_OPT1_S_REP_EATER_유 AT %MW10205.6 : BOOL; (* S368 M 차종 OPT1 S REP EATER 유 *)
    S368_M_차종_OPT1_VAN_무 AT %MW10205.9 : BOOL; (* S368 M 차종 OPT1 VAN 무 *)
    S368_M_차종_OPT1_VAN_유 AT %MW10205.8 : BOOL; (* S368 M 차종 OPT1 VAN 유 *)
    S368_M_차종_OPT1_슬라이딩_무 AT %MW10205.1 : BOOL; (* S368 M 차종 OPT1 슬라이딩 무 *)
    S368_M_차종_OPT1_슬라이딩_유 AT %MW10205.0 : BOOL; (* S368 M 차종 OPT1 슬라이딩 유 *)
    S368_M_차종_OPT1_폴딩_무 AT %MW10205.5 : BOOL; (* S368 M 차종 OPT1 폴딩 무 *)
    S368_M_차종_OPT1_폴딩_유 AT %MW10205.4 : BOOL; (* S368 M 차종 OPT1 폴딩 유 *)
    S368_M_차종_OPT2_SP_WORD1 AT %MW10206 : WORD; (* S368 M 차종 OPT2 SP WORD1 *)
    S368_M_차종_OPT3_SP_WORD2 AT %MW10207 : WORD; (* S368 M 차종 OPT3 SP WORD2 *)
    S368_M_차종_OPT4_SP_WORD3 AT %MW10208 : WORD; (* S368 M 차종 OPT4 SP WORD3 *)
    S368_M_차종_OPT5_SP_WORD4 AT %MW10209 : WORD; (* S368 M 차종 OPT5 SP WORD4 *)
    S368_M_차종_SP1 AT %MW10210.0 : BOOL; (* S368 M 차종 SP1 *)
    S368_M_차종_SP2 AT %MW10210.1 : BOOL; (* S368 M 차종 SP2 *)
    S368_M_차종_SP3 AT %MW10210.2 : BOOL; (* S368 M 차종 SP3 *)
    S368_M_차종_SP4 AT %MW10210.3 : BOOL; (* S368 M 차종 SP4 *)
    S368_M_차종_SP5 AT %MW10210.4 : BOOL; (* S368 M 차종 SP5 *)
    S368_M_차종_SP6 AT %MW10210.5 : BOOL; (* S368 M 차종 SP6 *)
    S368_M_차종_SP7 AT %MW10210.6 : BOOL; (* S368 M 차종 SP7 *)
    S368_M_차종_SP8 AT %MW10210.7 : BOOL; (* S368 M 차종 SP8 *)
    S368_M_차종_SP9 AT %MW10210.15 : BOOL; (* S368 M 차종 SP9 *)
    S368_M_차종_공대차 AT %MW10210.12 : BOOL; (* S368 M 차종 공대차 *)
    S368_M_차종_공차 AT %MW10210.10 : BOOL; (* S368 M 차종 공차 *)
    S368_M_차종_불량대차 AT %MW10210.13 : BOOL; (* S368 M 차종 불량대차 *)
    S368_M_차종_불량차 AT %MW10210.11 : BOOL; (* S368 M 차종 불량차 *)
    S368_M_차종_비축 AT %MW10210.8 : BOOL; (* S368 M 차종 비축 *)
    S368_M_차종_취출대차 AT %MW10210.14 : BOOL; (* S368 M 차종 취출대차 *)
    S368_M_총괄_CP_이상 AT %MW4009.7 : BOOL; (* S368 CP OFF 이상 *)
    S368_M_총괄_CT_이상 AT %MW4010.4 : BOOL; (* S368   TACK TIME 이상 *)
    S368_M_총괄_EOCR_이상 AT %MW4009.8 : BOOL; (* S368_M_총괄_EOCR_이상 *)
    S368_M_총괄_INV_이상 AT %MW4009.9 : BOOL; (* S368_M_총괄_INV_이상 *)
    S368_M_총괄_LS_이상 AT %MW4009.15 : BOOL; (* S368 LS 이상 *)
    S368_M_총괄_MATCH_이상 AT %MW4010.0 : BOOL; (* S368 매트SW 이상 *)
    S368_M_총괄_MC_이상 AT %MW4009.13 : BOOL; (* S368_M_총괄_MC_이상 *)
    S368_M_총괄_MOTOR_이상 AT %MW4010.3 : BOOL; (* S368_M_총괄_MOTOR_이상 *)
    S368_M_총괄_NFB_이상 AT %MW4009.11 : BOOL; (* S368_M_총괄_NFB_이상 *)
    S368_M_총괄_ROBOT_이상 AT %MW4010.1 : BOOL; (* S368 ROBOT 이상 *)
    S368_M_총괄_SAFETY_이상 AT %MW4009.2 : BOOL; (* S368_M_총괄_SAFETY_이상 *)
    S368_M_총괄_SRV_이상 AT %MW4009.10 : BOOL; (* S368_M_총괄_SRV_이상 *)
    S368_M_총괄_공기압_이상 AT %MW4009.3 : BOOL; (* S368 공기압 이상 *)
    S368_M_총괄_비상정지_이상 AT %MW4009.1 : BOOL; (* S368_M_총괄_비상정지_이상 *)
    S368_M_총괄_사양_이상 AT %MW4009.6 : BOOL; (* S368 사양 이상 *)
    S368_M_총괄_오버런_이상 AT %MW4009.12 : BOOL; (* S368_M_총괄_오버런_이상 *)
    S368_M_총괄_용접타점수_이상 AT %MW4010.2 : BOOL; (* S368 용접타점수 이상 *)
    S368_M_총괄_이상 AT %MW4009.0 : BOOL; (* S368_M_총괄_이상 *)
    S368_M_총괄_제품감지_이상 AT %MW4009.4 : BOOL; (* S368 제품감지 이상 *)
    S368_M_총괄_차종_이상 AT %MW4009.5 : BOOL; (* S368 차종 이상 *)
    S368_M_총괄_통신_이상 AT %MW4009.14 : BOOL; (* S368 통신이상 *)
    S368_RH_M_NODE_6_30_통신_이상 AT %MW4024.1 : BOOL;
    S368_전진_ON AT %MW4048.1 : BOOL; (* S368_전진_ON *)
    S368_후진_ON AT %MW4048.2 : BOOL; (* S368_후진_ON *)
    S369_1_M_BYPASS_보조 AT %MW4503.15 : BOOL; (* S369 1 M BYPASS 보조 *)
    S369_1_M_CTIME_OVER_ALRAM AT %MW4507.14 : BOOL; (* S369_1_M_CTIME_OVER_ALRAM *)
    S369_1_M_CTIME_OVER_MUTE AT %MW4507.13 : BOOL; (* S369_1_M_CTIME_OVER_MUTE *)
    S369_1_M_DATA_삭제_PLS AT %MW9018.0 : BOOL; (* S369_1 M DATA 삭제 PLS *)
    S369_1_M_DATA_삭제_SIGN AT %MW9018.1 : BOOL; (* S369_1 M DATA 삭제 SIGN *)
    S369_1_M_DATA_삭제_완료 AT %MW9018.2 : BOOL; (* S369_1 M DATA 삭제 완료 *)
    S369_1_M_LC_정상 AT %MW4507.5 : BOOL; (* S369_1_M_LC_정상 *)
    S369_1_M_MAT_정상 AT %MW4507.6 : BOOL; (* S369_1_M_MAT_정상 *)
    S369_1_M_NODE_6_40_통신_이상 AT %MW4524.0 : BOOL;
    S369_1_M_OP_ESTOP_NORMAL AT %MW4507.1 : BOOL; (* S369_1_M_OP_ESTOP_NORMAL *)
    S369_1_M_R369_1_안착완료 AT %MW4501.1 : BOOL;
    S369_1_M_R369_2_DATA_전송_MEMO AT %MW9018.8 : BOOL; (* S369_1 M R369 2 DATA 전송 MEMO *)
    S369_1_M_R369_2_DATA_전송_PLS AT %MW9018.9 : BOOL; (* S369_1 M R369 2 DATA 전송 PLS *)
    S369_1_M_R369_2_DATA_전송_SIGN AT %MW9018.10 : BOOL; (* S369_1 M R369 2 DATA 전송 SIGN *)
    S369_1_M_R369_2_DATA_전송_완료 AT %MW9018.11 : BOOL; (* S369_1 M R369 2 DATA 전송 완료 *)
    S369_1_M_R369_2_ROOF_취출가능 AT %MW4504.9 : BOOL;
    S369_1_M_R369_2_언로딩완료 AT %MW4501.2 : BOOL;
    S369_1_M_ROOF_안착가능 AT %MW4504.8 : BOOL;
    S369_1_M_ROOF_제품감지_무 AT %MW4501.6 : BOOL;
    S369_1_M_ROOF_제품감지_유 AT %MW4501.5 : BOOL;
    S369_1_M_ROOF_제품감지_이상 AT %MW4514.0 : BOOL;
    S369_1_M_S102_간섭무 AT %MW4504.2 : BOOL; (* S369_1_M_S102_간섭무 *)
    S369_1_M_SAFETY_불간섭 AT %MW4504.4 : BOOL; (* S369_1_M_SAFETY_불간섭 *)
    S369_1_M_SEMI_자동모드 AT %MW4500.2 : BOOL; (* S369_1_M_SEMI_자동모드 *)
    S369_1_M_SEQ AT %MW10220 : WORD; (* S369 1 M SEQ *)
    S369_1_M_VIN_NO_1_2 AT %MW10231 : WORD; (* S369 1 M VIN NO 1 2 *)
    S369_1_M_VIN_NO_3_4 AT %MW10232 : WORD; (* S369 1 M VIN NO 3 4 *)
    S369_1_M_VIN_NO_5_6 AT %MW10233 : WORD; (* S369 1 M VIN NO 5 6 *)
    S369_1_M_VIN_NO_7_8 AT %MW10234 : WORD; (* S369 1 M VIN NO 7 8 *)
    S369_1_M_VIN_NO_9_10 AT %MW10235 : WORD; (* S369 1 M VIN NO 9 10 *)
    S369_1_M_공정_SAFETY_NORMAL AT %MW4507.7 : BOOL; (* S369_1_M_공정_SAFETY_NORMAL *)
    S369_1_M_공정_불간섭 AT %MW4504.1 : BOOL; (* S369_1_M_공정_불간섭 *)
    S369_1_M_공정_원위치 AT %MW4504.0 : BOOL; (* S369_1_M_공정_원위치 *)
    S369_1_M_공정_제품감지_무 AT %MW4501.4 : BOOL; (* S369_1_M_공정_제품감지_무 *)
    S369_1_M_공정_제품감지_유 AT %MW4501.3 : BOOL; (* S369_1_M_공정_제품감지_유 *)
    S369_1_M_공정_차종_무 AT %MW4502.1 : BOOL; (* S369_1_M_공정_차종_무 *)
    S369_1_M_공정_차종_유 AT %MW4502.0 : BOOL; (* S369_1_M_공정_차종_유 *)
    S369_1_M_부저_정지_보조 AT %MW4500.11 : BOOL; (* S369_1_M_부저_정지_보조 *)
    S369_1_M_수동모드 AT %MW4500.3 : BOOL; (* S369-1 선택 수동모드 *)
    S369_1_M_썬루프_제품감지_무 AT %MW4501.8 : BOOL;
    S369_1_M_썬루프_제품감지_유 AT %MW4501.7 : BOOL;
    S369_1_M_썬루프_제품감지_이상 AT %MW4514.1 : BOOL;
    S369_1_M_운전준비_ON AT %MW4500.0 : BOOL; (* S369-1 운전준비 ON *)
    S369_1_M_이상_리셋_보조 AT %MW4500.10 : BOOL; (* S369_1_M_이상_리셋_보조 *)
    S369_1_M_자동_START AT %MW4500.5 : BOOL; (* S369-1 자동운전중 *)
    S369_1_M_자동_운전중 AT %MW4500.4 : BOOL; (* S369-1 자동운전중 *)
    S369_1_M_자동모드 AT %MW4500.1 : BOOL; (* S369-1 선택 자동모드 *)
    S369_1_M_작업_완료 AT %MW4501.0 : BOOL; (* S369_1_M_작업_완료 *)
    S369_1_M_작업완료_SET_PLS AT %MW4500.8 : BOOL; (* S369 1 M 작업완료 SET PLS *)
    S369_1_M_작업완료_리셋_PLS AT %MW4500.9 : BOOL; (* S369 1 M 작업완료 리셋 PLS *)
    S369_1_M_차종1_AX AT %MW10221.0 : BOOL; (* S369 1 M 차종1 AX *)
    S369_1_M_차종1_B AT %MW10221.1 : BOOL; (* S369 1 M 차종1 B *)
    S369_1_M_차종1_C AT %MW10221.2 : BOOL; (* S369 1 M 차종1 C *)
    S369_1_M_차종1_D AT %MW10221.3 : BOOL; (* S369 1 M 차종1 D *)
    S369_1_M_차종1_E AT %MW10221.4 : BOOL; (* S369 1 M 차종1 E *)
    S369_1_M_차종1_F AT %MW10221.5 : BOOL; (* S369 1 M 차종1 F *)
    S369_1_M_차종1_G AT %MW10221.6 : BOOL; (* S369 1 M 차종1 G *)
    S369_1_M_차종1_H AT %MW10221.7 : BOOL; (* S369 1 M 차종1 H *)
    S369_1_M_차종2_3DR AT %MW10221.8 : BOOL; (* S369 1 M 차종2 3DR *)
    S369_1_M_차종2_4DR AT %MW10221.9 : BOOL; (* S369 1 M 차종2 4DR *)
    S369_1_M_차종2_5DR AT %MW10221.10 : BOOL; (* S369 1 M 차종2 5DR *)
    S369_1_M_차종2_SP1 AT %MW10221.12 : BOOL; (* S369 1 M 차종2 SP1 *)
    S369_1_M_차종2_SP2 AT %MW10221.13 : BOOL; (* S369 1 M 차종2 SP2 *)
    S369_1_M_차종2_WGN AT %MW10221.11 : BOOL; (* S369 1 M 차종2 WGN *)
    S369_1_M_차종3_LHD AT %MW10221.14 : BOOL; (* S369 1 M 차종3 LHD *)
    S369_1_M_차종3_RHD AT %MW10221.15 : BOOL; (* S369 1 M 차종3 RHD *)
    S369_1_M_차종4_EEC AT %MW10222.3 : BOOL; (* S369 1 M 차종4 EEC *)
    S369_1_M_차종4_SP1 AT %MW10222.8 : BOOL; (* S369 1 M 차종4 SP1 *)
    S369_1_M_차종4_SP2 AT %MW10222.9 : BOOL; (* S369 1 M 차종4 SP2 *)
    S369_1_M_차종4_SP3 AT %MW10222.11 : BOOL; (* S369 1 M 차종4 SP3 *)
    S369_1_M_차종4_SP4 AT %MW10222.12 : BOOL; (* S369 1 M 차종4 SP4 *)
    S369_1_M_차종4_SP5 AT %MW10222.13 : BOOL; (* S369 1 M 차종4 SP5 *)
    S369_1_M_차종4_SP6 AT %MW10222.14 : BOOL; (* S369 1 M 차종4 SP6 *)
    S369_1_M_차종4_SP7 AT %MW10222.15 : BOOL; (* S369 1 M 차종4 SP7 *)
    S369_1_M_차종4_내수 AT %MW10222.0 : BOOL; (* S369 1 M 차종4 내수 *)
    S369_1_M_차종4_러시아 AT %MW10222.10 : BOOL; (* S369 1 M 차종4 러시아 *)
    S369_1_M_차종4_북미 AT %MW10222.2 : BOOL; (* S369 1 M 차종4 북미 *)
    S369_1_M_차종4_브라질 AT %MW10222.7 : BOOL; (* S369 1 M 차종4 브라질 *)
    S369_1_M_차종4_수출 AT %MW10222.1 : BOOL; (* S369 1 M 차종4 수출 *)
    S369_1_M_차종4_중국 AT %MW10222.6 : BOOL; (* S369 1 M 차종4 중국 *)
    S369_1_M_차종4_중동 AT %MW10222.5 : BOOL; (* S369 1 M 차종4 중동 *)
    S369_1_M_차종4_호주 AT %MW10222.4 : BOOL; (* S369 1 M 차종4 호주 *)
    S369_1_M_차종5_AT AT %MW10223.1 : BOOL; (* S369 1 M 차종5 AT *)
    S369_1_M_차종5_MT AT %MW10223.0 : BOOL; (* S369 1 M 차종5 MT *)
    S369_1_M_차종5_SP1 AT %MW10223.2 : BOOL; (* S369 1 M 차종5 SP1 *)
    S369_1_M_차종6_DSROOF AT %MW10223.6 : BOOL; (* S369 1 M 차종6 DSROOF *)
    S369_1_M_차종6_SP1 AT %MW10223.7 : BOOL; (* S369 1 M 차종6 SP1 *)
    S369_1_M_차종6_썬루프 AT %MW10223.4 : BOOL; (* S369 1 M 차종6 썬루프 *)
    S369_1_M_차종6_일반루프 AT %MW10223.3 : BOOL; (* S369 1 M 차종6 일반루프 *)
    S369_1_M_차종6_파노라마루프 AT %MW10223.5 : BOOL; (* S369 1 M 차종6 파노라마루프 *)
    S369_1_M_차종7_DSL AT %MW10223.9 : BOOL; (* S369 1 M 차종7 DSL *)
    S369_1_M_차종7_GSL AT %MW10223.8 : BOOL; (* S369 1 M 차종7 GSL *)
    S369_1_M_차종7_SP1 AT %MW10223.10 : BOOL; (* S369 1 M 차종7 SP1 *)
    S369_1_M_차종7_SP2 AT %MW10223.11 : BOOL; (* S369 1 M 차종7 SP2 *)
    S369_1_M_차종7_SP3 AT %MW10223.12 : BOOL; (* S369 1 M 차종7 SP3 *)
    S369_1_M_차종7_SP4 AT %MW10223.13 : BOOL; (* S369 1 M 차종7 SP4 *)
    S369_1_M_차종7_SP5 AT %MW10223.14 : BOOL; (* S369 1 M 차종7 SP5 *)
    S369_1_M_차종7_SP6 AT %MW10223.15 : BOOL; (* S369 1 M 차종7 SP6 *)
    S369_1_M_차종8_2WD AT %MW10224.0 : BOOL; (* S369 1 M 차종8 2WD *)
    S369_1_M_차종8_4WD AT %MW10224.1 : BOOL; (* S369 1 M 차종8 4WD *)
    S369_1_M_차종8_SP1 AT %MW10224.2 : BOOL; (* S369 1 M 차종8 SP1 *)
    S369_1_M_차종9_MPI AT %MW10224.3 : BOOL; (* S369 1 M 차종9 MPI *)
    S369_1_M_차종9_SP1 AT %MW10224.5 : BOOL; (* S369 1 M 차종9 SP1 *)
    S369_1_M_차종9_SP10 AT %MW10224.14 : BOOL; (* S369 1 M 차종9 SP10 *)
    S369_1_M_차종9_SP11 AT %MW10224.15 : BOOL; (* S369 1 M 차종9 SP11 *)
    S369_1_M_차종9_SP2 AT %MW10224.6 : BOOL; (* S369 1 M 차종9 SP2 *)
    S369_1_M_차종9_SP3 AT %MW10224.7 : BOOL; (* S369 1 M 차종9 SP3 *)
    S369_1_M_차종9_SP4 AT %MW10224.8 : BOOL; (* S369 1 M 차종9 SP4 *)
    S369_1_M_차종9_SP5 AT %MW10224.9 : BOOL; (* S369 1 M 차종9 SP5 *)
    S369_1_M_차종9_SP6 AT %MW10224.10 : BOOL; (* S369 1 M 차종9 SP6 *)
    S369_1_M_차종9_SP7 AT %MW10224.11 : BOOL; (* S369 1 M 차종9 SP7 *)
    S369_1_M_차종9_SP8 AT %MW10224.12 : BOOL; (* S369 1 M 차종9 SP8 *)
    S369_1_M_차종9_SP9 AT %MW10224.13 : BOOL; (* S369 1 M 차종9 SP9 *)
    S369_1_M_차종9_T_GDI AT %MW10224.4 : BOOL; (* S369 1 M 차종9 T GDI *)
    S369_1_M_차종_AS AT %MW10230.9 : BOOL; (* S369 1 M 차종 AS *)
    S369_1_M_차종_OPT1_R_RACK_무 AT %MW10225.3 : BOOL; (* S369 1 M 차종 OPT1 R RACK 무 *)
    S369_1_M_차종_OPT1_R_RACK_유 AT %MW10225.2 : BOOL; (* S369 1 M 차종 OPT1 R RACK 유 *)
    S369_1_M_차종_OPT1_SP1 AT %MW10225.10 : BOOL; (* S369 1 M 차종 OPT1 SP1 *)
    S369_1_M_차종_OPT1_SP2 AT %MW10225.11 : BOOL; (* S369 1 M 차종 OPT1 SP2 *)
    S369_1_M_차종_OPT1_SP3 AT %MW10225.12 : BOOL; (* S369 1 M 차종 OPT1 SP3 *)
    S369_1_M_차종_OPT1_SP4 AT %MW10225.13 : BOOL; (* S369 1 M 차종 OPT1 SP4 *)
    S369_1_M_차종_OPT1_SP5 AT %MW10225.14 : BOOL; (* S369 1 M 차종 OPT1 SP5 *)
    S369_1_M_차종_OPT1_SP6 AT %MW10225.15 : BOOL; (* S369 1 M 차종 OPT1 SP6 *)
    S369_1_M_차종_OPT1_S_REP_EATER_무 AT %MW10225.7 : BOOL; (* S369 1 M 차종 OPT1 S REP EATER 무 *)
    S369_1_M_차종_OPT1_S_REP_EATER_유 AT %MW10225.6 : BOOL; (* S369 1 M 차종 OPT1 S REP EATER 유 *)
    S369_1_M_차종_OPT1_VAN_무 AT %MW10225.9 : BOOL; (* S369 1 M 차종 OPT1 VAN 무 *)
    S369_1_M_차종_OPT1_VAN_유 AT %MW10225.8 : BOOL; (* S369 1 M 차종 OPT1 VAN 유 *)
    S369_1_M_차종_OPT1_슬라이딩_무 AT %MW10225.1 : BOOL; (* S369 1 M 차종 OPT1 슬라이딩 무 *)
    S369_1_M_차종_OPT1_슬라이딩_유 AT %MW10225.0 : BOOL; (* S369 1 M 차종 OPT1 슬라이딩 유 *)
    S369_1_M_차종_OPT1_폴딩_무 AT %MW10225.5 : BOOL; (* S369 1 M 차종 OPT1 폴딩 무 *)
    S369_1_M_차종_OPT1_폴딩_유 AT %MW10225.4 : BOOL; (* S369 1 M 차종 OPT1 폴딩 유 *)
    S369_1_M_차종_OPT2_SP_WORD1 AT %MW10226 : WORD; (* S369 1 M 차종 OPT2 SP WORD1 *)
    S369_1_M_차종_OPT3_SP_WORD2 AT %MW10227 : WORD; (* S369 1 M 차종 OPT3 SP WORD2 *)
    S369_1_M_차종_OPT4_SP_WORD3 AT %MW10228 : WORD; (* S369 1 M 차종 OPT4 SP WORD3 *)
    S369_1_M_차종_OPT5_SP_WORD4 AT %MW10229 : WORD; (* S369 1 M 차종 OPT5 SP WORD4 *)
    S369_1_M_차종_SP1 AT %MW10230.0 : BOOL; (* S369 1 M 차종 SP1 *)
    S369_1_M_차종_SP2 AT %MW10230.1 : BOOL; (* S369 1 M 차종 SP2 *)
    S369_1_M_차종_SP3 AT %MW10230.2 : BOOL; (* S369 1 M 차종 SP3 *)
    S369_1_M_차종_SP4 AT %MW10230.3 : BOOL; (* S369 1 M 차종 SP4 *)
    S369_1_M_차종_SP5 AT %MW10230.4 : BOOL; (* S369 1 M 차종 SP5 *)
    S369_1_M_차종_SP6 AT %MW10230.5 : BOOL; (* S369 1 M 차종 SP6 *)
    S369_1_M_차종_SP7 AT %MW10230.6 : BOOL; (* S369 1 M 차종 SP7 *)
    S369_1_M_차종_SP8 AT %MW10230.7 : BOOL; (* S369 1 M 차종 SP8 *)
    S369_1_M_차종_SP9 AT %MW10230.15 : BOOL; (* S369 1 M 차종 SP9 *)
    S369_1_M_차종_공대차 AT %MW10230.12 : BOOL; (* S369 1 M 차종 공대차 *)
    S369_1_M_차종_공차 AT %MW10230.10 : BOOL; (* S369 1 M 차종 공차 *)
    S369_1_M_차종_불량대차 AT %MW10230.13 : BOOL; (* S369 1 M 차종 불량대차 *)
    S369_1_M_차종_불량차 AT %MW10230.11 : BOOL; (* S369 1 M 차종 불량차 *)
    S369_1_M_차종_비축 AT %MW10230.8 : BOOL; (* S369 1 M 차종 비축 *)
    S369_1_M_차종_취출대차 AT %MW10230.14 : BOOL; (* S369 1 M 차종 취출대차 *)
    S369_1_M_총괄_CP_이상 AT %MW4509.7 : BOOL; (* S369-1 CP OFF 이상 *)
    S369_1_M_총괄_CT_이상 AT %MW4510.4 : BOOL; (* S369-1 TACK TIME 이상 *)
    S369_1_M_총괄_EOCR_이상 AT %MW4509.8 : BOOL; (* S369_1_M_총괄_EOCR_이상 *)
    S369_1_M_총괄_INV_이상 AT %MW4509.9 : BOOL; (* S369_1_M_총괄_INV_이상 *)
    S369_1_M_총괄_LS_이상 AT %MW4509.15 : BOOL; (* S369-1 LS 이상 *)
    S369_1_M_총괄_MATCH_이상 AT %MW4510.0 : BOOL; (* S369-1 매트SW 이상 *)
    S369_1_M_총괄_MC_이상 AT %MW4509.13 : BOOL; (* S369_1_M_총괄_MC_이상 *)
    S369_1_M_총괄_MOTOR_이상 AT %MW4510.3 : BOOL; (* S369_1_M_총괄_MOTOR_이상 *)
    S369_1_M_총괄_NFB_이상 AT %MW4509.11 : BOOL; (* S369_1_M_총괄_NFB_이상 *)
    S369_1_M_총괄_ROBOT_이상 AT %MW4510.1 : BOOL; (* S369-1 ROBOT 이상 *)
    S369_1_M_총괄_SAFETY_이상 AT %MW4509.2 : BOOL; (* S369_1_M_총괄_SAFETY_이상 *)
    S369_1_M_총괄_SRV_이상 AT %MW4509.10 : BOOL; (* S369_1_M_총괄_SRV_이상 *)
    S369_1_M_총괄_공기압_이상 AT %MW4509.3 : BOOL; (* S36-1 공기압 이상 *)
    S369_1_M_총괄_비상정지_이상 AT %MW4509.1 : BOOL; (* S369_1_M_총괄_비상정지_이상 *)
    S369_1_M_총괄_사양_이상 AT %MW4509.6 : BOOL; (* S369-1 사양 이상 *)
    S369_1_M_총괄_오버런_이상 AT %MW4509.12 : BOOL; (* S369_1_M_총괄_오버런_이상 *)
    S369_1_M_총괄_용접타점수_이상 AT %MW4510.2 : BOOL; (* S369-1 용접타점수 이상 *)
    S369_1_M_총괄_이상 AT %MW4509.0 : BOOL; (* S369_1_M_총괄_이상 *)
    S369_1_M_총괄_제품감지_이상 AT %MW4509.4 : BOOL; (* S369-1 제품감지 이상 *)
    S369_1_M_총괄_차종_이상 AT %MW4509.5 : BOOL; (* S369-1 차종 이상 *)
    S369_1_M_총괄_통신_이상 AT %MW4509.14 : BOOL; (* S369-1 통신이상 *)
    S369_HOME AT %MW5048.0 : BOOL; (* S369_HOME *)
    S369_LOAD_M_NODE_6_41_통신_이상 AT %MW5024.0 : BOOL;
    S369_M_CTIME_OVER_ALRAM AT %MW5007.14 : BOOL; (* S369_M_CTIME_OVER_ALRAM *)
    S369_M_CTIME_OVER_MUTE AT %MW5007.13 : BOOL; (* S369_M_CTIME_OVER_MUTE *)
    S369_M_LC_정상 AT %MW5007.5 : BOOL; (* S369_M_LC_정상 *)
    S369_M_LD_BYPASS_보조 AT %MW5003.14 : BOOL;
    S369_M_LD_CP_OFF AT %MW5017.0 : BOOL; (* S369_M_LD_CP_OFF *)
    S369_M_LD_EJECT_상승_LS_이상 AT %MW5100.5 : BOOL; (* S369_M_LD_EJECT_상승_LS_이상 *)
    S369_M_LD_EJECT_상승_보조 AT %MW5100.1 : BOOL; (* S369_M_LD_EJECT_상승_보조 *)
    S369_M_LD_EJECT_상승단 AT %MW5100.3 : BOOL; (* S369_M_LD_EJECT_상승단 *)
    S369_M_LD_EJECT_제품감지_이상 AT %MW5014.0 : BOOL; (* S369_M_LD_제품감지_이상 *)
    S369_M_LD_EJECT_조건 AT %MW5100.0 : BOOL; (* S369_M_LD_EJECT_조건 *)
    S369_M_LD_EJECT_하강_LS_이상 AT %MW5100.6 : BOOL; (* S369_M_LD_EJECT_하강_LS_이상 *)
    S369_M_LD_EJECT_하강_보조 AT %MW5100.2 : BOOL; (* S369_M_LD_EJECT_하강_보조 *)
    S369_M_LD_EJECT_하강단 AT %MW5100.4 : BOOL; (* S369_M_LD_EJECT_하강단 *)
    S369_M_LD_LH_LAT_전진_LS_이상 AT %MW5101.5 : BOOL; (* S369_M_LD_LH_LAT_전진_LS_이상 *)
    S369_M_LD_LH_LAT_전진_보조 AT %MW5101.1 : BOOL; (* S369_M_LD_LH_LAT_전진_보조 *)
    S369_M_LD_LH_LAT_전진단 AT %MW5101.3 : BOOL; (* S369_M_LD_LH_LAT_전진단 *)
    S369_M_LD_LH_LAT_조건 AT %MW5101.0 : BOOL; (* S369_M_LD_LH_LAT_조건 *)
    S369_M_LD_LH_LAT_후진_LS_이상 AT %MW5101.6 : BOOL; (* S369_M_LD_LH_LAT_후진_LS_이상 *)
    S369_M_LD_LH_LAT_후진_보조 AT %MW5101.2 : BOOL; (* S369_M_LD_LH_LAT_후진_보조 *)
    S369_M_LD_LH_LAT_후진단 AT %MW5101.4 : BOOL; (* S369_M_LD_LH_LAT_후진단 *)
    S369_M_LD_RH_LAT_전진_LS_이상 AT %MW5102.5 : BOOL; (* S369_M_LD_RH_LAT_전진_LS_이상 *)
    S369_M_LD_RH_LAT_전진_보조 AT %MW5102.1 : BOOL; (* S369_M_LD_RH_LAT_전진_보조 *)
    S369_M_LD_RH_LAT_전진단 AT %MW5102.3 : BOOL; (* S369_M_LD_RH_LAT_전진단 *)
    S369_M_LD_RH_LAT_조건 AT %MW5102.0 : BOOL; (* S369_M_LD_RH_LAT_조건 *)
    S369_M_LD_RH_LAT_후진_LS_이상 AT %MW5102.6 : BOOL; (* S369_M_LD_RH_LAT_후진_LS_이상 *)
    S369_M_LD_RH_LAT_후진_보조 AT %MW5102.2 : BOOL; (* S369_M_LD_RH_LAT_후진_보조 *)
    S369_M_LD_RH_LAT_후진단 AT %MW5102.4 : BOOL; (* S369_M_LD_RH_LAT_후진단 *)
    S369_M_LD_공기압_이상 AT %MW5013.0 : BOOL; (* S369_M_LD_공기압_이상 *)
    S369_M_LD_작업완료_SET_PLS AT %MW5000.6 : BOOL;
    S369_M_LD_작업완료_리셋_PLS AT %MW5000.7 : BOOL;
    S369_M_LD_차종_이상 AT %MW5015.0 : BOOL; (* S369_M_LD_차종_이상 *)
    S369_M_MAT_정상 AT %MW5007.6 : BOOL; (* S369_M_MAT_정상 *)
    S369_M_OP_ESTOP_NORMAL AT %MW5007.1 : BOOL; (* S369_M_OP_ESTOP_NORMAL *)
    S369_M_R308_3_언로딩가능 AT %MW5004.9 : BOOL;
    S369_M_R308_3_언로딩완료 AT %MW5001.5 : BOOL;
    S369_M_R308_3_클램프완료 AT %MW5001.4 : BOOL;
    S369_M_R308_3_클램프요구 AT %MW5004.11 : BOOL;
    S369_M_R308_3_행거안착가능 AT %MW5004.10 : BOOL;
    S369_M_R308_3_행거안착완료 AT %MW5001.3 : BOOL;
    S369_M_R369_2_로딩가능 AT %MW5004.8 : BOOL;
    S369_M_R369_2_로딩완료 AT %MW5001.2 : BOOL;
    S369_M_SAFETY_불간섭 AT %MW5004.4 : BOOL; (* S369_M_SAFETY_불간섭 *)
    S369_M_SEMI_자동모드 AT %MW5000.2 : BOOL; (* S369_M_SEMI_자동모드 *)
    S369_M_SERVO_DRIVE_통신이상 AT %MW5024.8 : BOOL;
    S369_M_SRV_NFB_OFF AT %MW5021.0 : BOOL; (* S369_M_SRV_NFB_OFF *)
    S369_M_SRV_이상 AT %MW5020.0 : BOOL; (* S369_M_SRV_이상 *)
    S369_M_UD_BYPASS_보조 AT %MW5003.15 : BOOL; (* S369 M BYPASS 보조 *)
    S369_M_UD_CP_OFF AT %MW5017.1 : BOOL; (* S369_M_UD_CP_OFF *)
    S369_M_UD_DOCK_CLP_전진_LS_이상 AT %MW5111.5 : BOOL; (* S369_M_UD_DOCK_CLP_전진_LS_이상 *)
    S369_M_UD_DOCK_CLP_전진_보조 AT %MW5111.1 : BOOL; (* S369_M_UD_DOCK_CLP_전진_보조 *)
    S369_M_UD_DOCK_CLP_전진단 AT %MW5111.3 : BOOL; (* S369_M_UD_DOCK_CLP_전진단 *)
    S369_M_UD_DOCK_CLP_조건 AT %MW5111.0 : BOOL; (* S369_M_UD_DOCK_CLP_조건 *)
    S369_M_UD_DOCK_CLP_후진_LS_이상 AT %MW5111.6 : BOOL; (* S369_M_UD_DOCK_CLP_후진_LS_이상 *)
    S369_M_UD_DOCK_CLP_후진_보조 AT %MW5111.2 : BOOL; (* S369_M_UD_DOCK_CLP_후진_보조 *)
    S369_M_UD_DOCK_CLP_후진단 AT %MW5111.4 : BOOL; (* S369_M_UD_DOCK_CLP_후진단 *)
    S369_M_UD_EJECT_상승_LS_이상 AT %MW5108.5 : BOOL; (* S369_M_UD_EJECT_상승_LS_이상 *)
    S369_M_UD_EJECT_상승_보조 AT %MW5108.1 : BOOL; (* S369_M_UD_EJECT_상승_보조 *)
    S369_M_UD_EJECT_상승단 AT %MW5108.3 : BOOL; (* S369_M_UD_EJECT_상승단 *)
    S369_M_UD_EJECT_제품감지_이상 AT %MW5014.1 : BOOL; (* S369_M_UD_제품감지_이상 *)
    S369_M_UD_EJECT_조건 AT %MW5108.0 : BOOL; (* S369_M_UD_EJECT_조건 *)
    S369_M_UD_EJECT_하강_LS_이상 AT %MW5108.6 : BOOL; (* S369_M_UD_EJECT_하강_LS_이상 *)
    S369_M_UD_EJECT_하강_보조 AT %MW5108.2 : BOOL; (* S369_M_UD_EJECT_하강_보조 *)
    S369_M_UD_EJECT_하강단 AT %MW5108.4 : BOOL; (* S369_M_UD_EJECT_하강단 *)
    S369_M_UD_LH_LAT_전진_LS_이상 AT %MW5109.5 : BOOL; (* S369_M_UD_LH_LAT_전진_LS_이상 *)
    S369_M_UD_LH_LAT_전진_보조 AT %MW5109.1 : BOOL; (* S369_M_UD_LH_LAT_전진_보조 *)
    S369_M_UD_LH_LAT_전진단 AT %MW5109.3 : BOOL; (* S369_M_UD_LH_LAT_전진단 *)
    S369_M_UD_LH_LAT_조건 AT %MW5109.0 : BOOL; (* S369_M_UD_LH_LAT_조건 *)
    S369_M_UD_LH_LAT_후진_LS_이상 AT %MW5109.6 : BOOL; (* S369_M_UD_LH_LAT_후진_LS_이상 *)
    S369_M_UD_LH_LAT_후진_보조 AT %MW5109.2 : BOOL; (* S369_M_UD_LH_LAT_후진_보조 *)
    S369_M_UD_LH_LAT_후진단 AT %MW5109.4 : BOOL; (* S369_M_UD_LH_LAT_후진단 *)
    S369_M_UD_RH_LAT_전진_LS_이상 AT %MW5110.5 : BOOL; (* S369_M_UD_RH_LAT_전진_LS_이상 *)
    S369_M_UD_RH_LAT_전진_보조 AT %MW5110.1 : BOOL; (* S369_M_UD_RH_LAT_전진_보조 *)
    S369_M_UD_RH_LAT_전진단 AT %MW5110.3 : BOOL; (* S369_M_UD_RH_LAT_전진단 *)
    S369_M_UD_RH_LAT_조건 AT %MW5110.0 : BOOL; (* S369_M_UD_RH_LAT_조건 *)
    S369_M_UD_RH_LAT_후진_LS_이상 AT %MW5110.6 : BOOL; (* S369_M_UD_RH_LAT_후진_LS_이상 *)
    S369_M_UD_RH_LAT_후진_보조 AT %MW5110.2 : BOOL; (* S369_M_UD_RH_LAT_후진_보조 *)
    S369_M_UD_RH_LAT_후진단 AT %MW5110.4 : BOOL; (* S369_M_UD_RH_LAT_후진단 *)
    S369_M_UD_공기압_이상 AT %MW5013.1 : BOOL; (* S369_M_UD_공기압_이상 *)
    S369_M_UD_작업완료_SET_PLS AT %MW5000.8 : BOOL; (* S369 M 작업완료 SET PLS *)
    S369_M_UD_작업완료_리셋_PLS AT %MW5000.9 : BOOL; (* S369 M 작업완료 리셋 PLS *)
    S369_M_UD_차종_이상 AT %MW5015.1 : BOOL; (* S369_M_UD_차종_이상 *)
    S369_M_공정_SAFETY_NORMAL AT %MW5007.7 : BOOL; (* S369_M_공정_SAFETY_NORMAL *)
    S369_M_동작_선택_1 AT %MW5040.0 : BOOL; (* S369_M_동작_선택_1 *)
    S369_M_동작_선택_10 AT %MW5040.9 : BOOL; (* S369_M_동작_선택_10 *)
    S369_M_동작_선택_11 AT %MW5040.10 : BOOL; (* S369_M_동작_선택_11 *)
    S369_M_동작_선택_12 AT %MW5040.11 : BOOL; (* S369_M_동작_선택_12 *)
    S369_M_동작_선택_13 AT %MW5040.12 : BOOL; (* S369_M_동작_선택_13 *)
    S369_M_동작_선택_14 AT %MW5040.13 : BOOL; (* S369_M_동작_선택_14 *)
    S369_M_동작_선택_15 AT %MW5040.14 : BOOL; (* S369_M_동작_선택_15 *)
    S369_M_동작_선택_16 AT %MW5040.15 : BOOL; (* S369_M_동작_선택_16 *)
    S369_M_동작_선택_17 AT %MW5041.0 : BOOL; (* S369_M_동작_선택_17 *)
    S369_M_동작_선택_18 AT %MW5041.1 : BOOL; (* S369_M_동작_선택_18 *)
    S369_M_동작_선택_19 AT %MW5041.2 : BOOL; (* S369_M_동작_선택_19 *)
    S369_M_동작_선택_2 AT %MW5040.1 : BOOL; (* S369_M_동작_선택_2 *)
    S369_M_동작_선택_20 AT %MW5041.3 : BOOL; (* S369_M_동작_선택_20 *)
    S369_M_동작_선택_21 AT %MW5041.4 : BOOL; (* S369_M_동작_선택_21 *)
    S369_M_동작_선택_22 AT %MW5041.5 : BOOL; (* S369_M_동작_선택_22 *)
    S369_M_동작_선택_23 AT %MW5041.6 : BOOL; (* S369_M_동작_선택_23 *)
    S369_M_동작_선택_24 AT %MW5041.7 : BOOL; (* S369_M_동작_선택_24 *)
    S369_M_동작_선택_25 AT %MW5041.8 : BOOL; (* S369_M_동작_선택_25 *)
    S369_M_동작_선택_26 AT %MW5041.9 : BOOL; (* S369_M_동작_선택_26 *)
    S369_M_동작_선택_27 AT %MW5041.10 : BOOL; (* S369_M_동작_선택_27 *)
    S369_M_동작_선택_28 AT %MW5041.11 : BOOL; (* S369_M_동작_선택_28 *)
    S369_M_동작_선택_29 AT %MW5041.12 : BOOL; (* S369_M_동작_선택_29 *)
    S369_M_동작_선택_3 AT %MW5040.2 : BOOL; (* S369_M_동작_선택_3 *)
    S369_M_동작_선택_30 AT %MW5041.13 : BOOL; (* S369_M_동작_선택_30 *)
    S369_M_동작_선택_31 AT %MW5041.14 : BOOL; (* S369_M_동작_선택_31 *)
    S369_M_동작_선택_32 AT %MW5041.15 : BOOL; (* S369_M_동작_선택_32 *)
    S369_M_동작_선택_4 AT %MW5040.3 : BOOL; (* S369_M_동작_선택_4 *)
    S369_M_동작_선택_5 AT %MW5040.4 : BOOL; (* S369_M_동작_선택_5 *)
    S369_M_동작_선택_6 AT %MW5040.5 : BOOL; (* S369_M_동작_선택_6 *)
    S369_M_동작_선택_7 AT %MW5040.6 : BOOL; (* S369_M_동작_선택_7 *)
